THIS^.testValueIsNaN(THIS^.NAN);
THIS^.testValueIsNaN(THIS^.INF);
THIS^.testValueIsNaN(THIS^.MINUS_INF);
THIS^.testValueIsNaN(THIS^.MAX_NON_SPECIAL);
THIS^.testValueIsNaN(THIS^.MIN_NON_SPECIAL);
THIS^.testValueIsNaN(THIS^.ZERO);
THIS^.testValueIsNaN(THIS^.MINUS_ZERO);
THIS^.testValueIsNaN(THIS^.MAX_SUBNORMAL);
THIS^.testValueIsNaN(THIS^.MIN_SUBNORMAL);
THIS^.testValueIsNaN(THIS^.SMALLEST_NEGATIVE_SUBNORMAL);
THIS^.testValueIsNaN(THIS^.SMALLEST_POSITIVE_SUBNORMAL);
THIS^.testValueIsNaN(THIS^.ONE_PERCENT);
THIS^.testValueIsNaN(THIS^.ONE_PERMILLE);
THIS^.testValueIsNaN(THIS^.MINUS_ONE_PERCENT);
THIS^.testValueIsNaN(THIS^.MINUS_ONE_PERMILLE);

TcUnit.TEST_FINISHED();
END_METHOD

(*

short summary
==================
This test method tests ``assert.float.double.valueIsNegativeInfinite``
method of CNM_AssertionInterfaces library with various inputs

.. <legal notes>

legal notes
=================
| SPDX-FileCopyrightText: © 2022 ekvip automation GmbH <info@ekvip.de>
| SPDX-License-Identifier: Apache-2.0
| For details check: Apache-2.0_

.. _Apache-2.0: https://www.apache.org/licenses/LICENSE-2.0

.. </legal notes>

*)

METHOD runValueIsNegativeInfiniteTests
RETURN (NOT TcUnit.TEST_ORDERED(THIS^.getTestNameFor('valueIsNegativeInfinite')));

THIS^.testValueIsNegativeInfinite(THIS^.NAN);
THIS^.testValueIsNegativeInfinite(THIS^.INF);
THIS^.testValueIsNegativeInfinite(THIS^.MINUS_INF);
THIS^.testValueIsNegativeInfinite(THIS^.MAX_NON_SPECIAL);
THIS^.testValueIsNegativeInfinite(THIS^.MIN_NON_SPECIAL);
THIS^.testValueIsNegativeInfinite(THIS^.ZERO);
THIS^.testValueIsNegativeInfinite(THIS^.MINUS_ZERO);
THIS^.testValueIsNegativeInfinite(THIS^.MAX_SUBNORMAL);
THIS^.testValueIsNegativeInfinite(THIS^.MIN_SUBNORMAL);
THIS^.testValueIsNegativeInfinite(THIS^.SMALLEST_NEGATIVE_SUBNORMAL);
THIS^.testValueIsNegativeInfinite(THIS^.SMALLEST_POSITIVE_SUBNORMAL);
THIS^.testValueIsNegativeInfinite(THIS^.ONE_PERCENT);
THIS^.testValueIsNegativeInfinite(THIS^.ONE_PERMILLE);
THIS^.testValueIsNegativeInfinite(THIS^.MINUS_ONE_PERCENT);
THIS^.testValueIsNegativeInfinite(THIS^.MINUS_ONE_PERMILLE);

TcUnit.TEST_FINISHED();
END_METHOD

(*

short summary
==================
This test method tests ``assert.float.double.valueIsNegative``
method of CNM_AssertionInterfaces library with various inputs

.. <legal notes>

legal notes
=================
| SPDX-FileCopyrightText: © 2022 ekvip automation GmbH <info@ekvip.de>
| SPDX-License-Identifier: Apache-2.0
| For details check: Apache-2.0_

.. _Apache-2.0: https://www.apache.org/licenses/LICENSE-2.0

.. </legal notes>

*)

METHOD runValueIsNegativeTests
RETURN (NOT TcUnit.TEST_ORDERED(THIS^.getTestNameFor('valueIsNegative')));

THIS^.testValueIsNegative(THIS^.NAN);
THIS^.testValueIsNegative(THIS^.INF);
THIS^.testValueIsNegative(THIS^.MINUS_INF);
THIS^.testValueIsNegative(THIS^.MAX_NON_SPECIAL);
THIS^.testValueIsNegative(THIS^.MIN_NON_SPECIAL);
THIS^.testValueIsNegative(THIS^.ZERO);
THIS^.testValueIsNegative(THIS^.MINUS_ZERO);
THIS^.testValueIsNegative(THIS^.MAX_SUBNORMAL);
THIS^.testValueIsNegative(THIS^.MIN_SUBNORMAL);
THIS^.testValueIsNegative(THIS^.SMALLEST_NEGATIVE_SUBNORMAL);
THIS^.testValueIsNegative(THIS^.SMALLEST_POSITIVE_SUBNORMAL);
THIS^.testValueIsNegative(THIS^.ONE_PERCENT);
THIS^.testValueIsNegative(THIS^.ONE_PERMILLE);
THIS^.testValueIsNegative(THIS^.MINUS_ONE_PERCENT);
THIS^.testValueIsNegative(THIS^.MINUS_ONE_PERMILLE);

TcUnit.TEST_FINISHED();
END_METHOD

(*

short summary
==================
This test method tests ``assert.float.double.valueIsNegativeZero``
method of CNM_AssertionInterfaces library with various inputs

.. <legal notes>

legal notes
=================
| SPDX-FileCopyrightText: © 2022 ekvip automation GmbH <info@ekvip.de>
| SPDX-License-Identifier: Apache-2.0
| For details check: Apache-2.0_

.. _Apache-2.0: https://www.apache.org/licenses/LICENSE-2.0

.. </legal notes>

*)

METHOD runValueIsNegativeZeroTests
RETURN (NOT TcUnit.TEST_ORDERED(THIS^.getTestNameFor('valueIsNegativeZero')));

THIS^.testValueIsNegativeZero(THIS^.NAN);
THIS^.testValueIsNegativeZero(THIS^.INF);
THIS^.testValueIsNegativeZero(THIS^.MINUS_INF);
THIS^.testValueIsNegativeZero(THIS^.MAX_NON_SPECIAL);
THIS^.testValueIsNegativeZero(THIS^.MIN_NON_SPECIAL);
THIS^.testValueIsNegativeZero(THIS^.ZERO);
THIS^.testValueIsNegativeZero(THIS^.MINUS_ZERO);
THIS^.testValueIsNegativeZero(THIS^.MAX_SUBNORMAL);
THIS^.testValueIsNegativeZero(THIS^.MIN_SUBNORMAL);
THIS^.testValueIsNegativeZero(THIS^.SMALLEST_NEGATIVE_SUBNORMAL);
THIS^.testValueIsNegativeZero(THIS^.SMALLEST_POSITIVE_SUBNORMAL);
THIS^.testValueIsNegativeZero(THIS^.ONE_PERCENT);
THIS^.testValueIsNegativeZero(THIS^.ONE_PERMILLE);
THIS^.testValueIsNegativeZero(THIS^.MINUS_ONE_PERCENT);
THIS^.testValueIsNegativeZero(THIS^.MINUS_ONE_PERMILLE);

TcUnit.TEST_FINISHED();
END_METHOD

(*

short summary
==================
This test method tests ``assert.float.double.valueIsNormal``
method of CNM_AssertionInterfaces library with various inputs

.. <legal notes>

legal notes
=================
| SPDX-FileCopyrightText: © 2022 ekvip automation GmbH <info@ekvip.de>
| SPDX-License-Identifier: Apache-2.0
| For details check: Apache-2.0_

.. _Apache-2.0: https://www.apache.org/licenses/LICENSE-2.0

.. </legal notes>

*)

METHOD runValueIsNormalTests
RETURN (NOT TcUnit.TEST_ORDERED(THIS^.getTestNameFor('valueIsNormal')));

THIS^.testValueIsNormal(THIS^.NAN);
THIS^.testValueIsNormal(THIS^.INF);
THIS^.testValueIsNormal(THIS^.MINUS_INF);
THIS^.testValueIsNormal(THIS^.MAX_NON_SPECIAL);
THIS^.testValueIsNormal(THIS^.MIN_NON_SPECIAL);
THIS^.testValueIsNormal(THIS^.ZERO);
THIS^.testValueIsNormal(THIS^.MINUS_ZERO);
THIS^.testValueIsNormal(THIS^.MAX_SUBNORMAL);
THIS^.testValueIsNormal(THIS^.MIN_SUBNORMAL);
THIS^.testValueIsNormal(THIS^.SMALLEST_NEGATIVE_SUBNORMAL);
THIS^.testValueIsNormal(THIS^.SMALLEST_POSITIVE_SUBNORMAL);
THIS^.testValueIsNormal(THIS^.ONE_PERCENT);
THIS^.testValueIsNormal(THIS^.ONE_PERMILLE);
THIS^.testValueIsNormal(THIS^.MINUS_ONE_PERCENT);
THIS^.testValueIsNormal(THIS^.MINUS_ONE_PERMILLE);

TcUnit.TEST_FINISHED();
END_METHOD

(*

short summary
==================
This test method tests ``assert.float.double.valueIsNotEqualTo``
method of CNM_AssertionInterfaces library with various inputs

.. <legal notes>

legal notes
=================
| SPDX-FileCopyrightText: © 2022 ekvip automation GmbH <info@ekvip.de>
| SPDX-License-Identifier: Apache-2.0
| For details check: Apache-2.0_

.. _Apache-2.0: https://www.apache.org/licenses/LICENSE-2.0

.. </legal notes>

*)

METHOD runValueIsNotEqualToTests
RETURN (NOT TcUnit.TEST_ORDERED(THIS^.getTestNameFor('valueIsNotEqualTo')));

THIS^.testValueIsNotEqualTo(
	valueToTest := THIS^.NAN,
	unexpectedValue := THIS^.ONE_PERCENT,
	tolerance := THIS^.ONE_PERMILLE
);

THIS^.testValueIsNotEqualTo(
	valueToTest := THIS^.ONE_PERCENT,
	unexpectedValue := THIS^.NAN,
	tolerance := THIS^.ONE_PERMILLE
);

THIS^.testValueIsNotEqualTo(
	valueToTest := THIS^.ONE_PERCENT,
	unexpectedValue := THIS^.ONE_PERCENT,
	tolerance := THIS^.NAN
);

THIS^.testValueIsNotEqualTo(
	valueToTest := THIS^.NAN,
	unexpectedValue := THIS^.NAN,
	tolerance := THIS^.ONE_PERCENT
);

THIS^.testValueIsNotEqualTo(
	valueToTest := THIS^.NAN,
	unexpectedValue := THIS^.NAN,
	tolerance := THIS^.NAN
);

THIS^.testValueIsNotEqualTo(
	valueToTest := THIS^.INF,
	unexpectedValue := THIS^.ONE_PERCENT,
	tolerance := THIS^.ONE_PERMILLE
);

THIS^.testValueIsNotEqualTo(
	valueToTest := THIS^.ONE_PERCENT,
	unexpectedValue := THIS^.INF,
	tolerance := THIS^.ONE_PERMILLE
);

THIS^.testValueIsNotEqualTo(
	valueToTest := THIS^.ONE_PERCENT,
	unexpectedValue := THIS^.ONE_PERCENT,
	tolerance := THIS^.INF
);

THIS^.testValueIsNotEqualTo(
	valueToTest := THIS^.INF,
	unexpectedValue := THIS^.INF,
	tolerance := THIS^.ONE_PERCENT
);

THIS^.testValueIsNotEqualTo(
	valueToTest := THIS^.INF,
	unexpectedValue := THIS^.INF,
	tolerance := THIS^.INF
);

THIS^.testValueIsNotEqualTo(
	valueToTest := THIS^.INF,
	unexpectedValue := THIS^.MINUS_INF,
	tolerance := THIS^.INF
);

THIS^.testValueIsNotEqualTo(
	valueToTest := THIS^.MINUS_INF,
	unexpectedValue := THIS^.ONE_PERCENT,
	tolerance := THIS^.ONE_PERMILLE
);

THIS^.testValueIsNotEqualTo(
	valueToTest := THIS^.ONE_PERCENT,
	unexpectedValue := THIS^.MINUS_INF,
	tolerance := THIS^.ONE_PERMILLE
);

THIS^.testValueIsNotEqualTo(
	valueToTest := THIS^.ONE_PERCENT,
	unexpectedValue := THIS^.ONE_PERCENT,
	tolerance := THIS^.MINUS_INF
);

THIS^.testValueIsNotEqualTo(
	valueToTest := THIS^.MINUS_INF,
	unexpectedValue := THIS^.MINUS_INF,
	tolerance := THIS^.ONE_PERCENT
);

THIS^.testValueIsNotEqualTo(
	valueToTest := THIS^.MINUS_INF,
	unexpectedValue := THIS^.MINUS_INF,
	tolerance := THIS^.MINUS_INF
);

THIS^.testValueIsNotEqualTo(
	valueToTest := THIS^.INF,
	unexpectedValue := THIS^.MINUS_INF,
	tolerance := THIS^.INF
);

THIS^.testValueIsNotEqualTo(
	valueToTest := THIS^.MINUS_ZERO,
	unexpectedValue := THIS^.SMALLEST_POSITIVE_SUBNORMAL,
	tolerance := THIS^.ONE_PERMILLE
);

THIS^.testValueIsNotEqualTo(
	valueToTest := THIS^.SMALLEST_POSITIVE_SUBNORMAL,
	unexpectedValue := THIS^.MINUS_ZERO,
	tolerance := THIS^.ONE_PERMILLE
);

THIS^.testValueIsNotEqualTo(
	valueToTest := THIS^.SMALLEST_POSITIVE_SUBNORMAL,
	unexpectedValue := THIS^.SMALLEST_POSITIVE_SUBNORMAL,
	tolerance := THIS^.MINUS_ZERO
);

THIS^.testValueIsNotEqualTo(
	valueToTest := THIS^.MINUS_ZERO,
	unexpectedValue := THIS^.MINUS_ZERO,
	tolerance := THIS^.SMALLEST_POSITIVE_SUBNORMAL
);

THIS^.testValueIsNotEqualTo(
	valueToTest := THIS^.MINUS_ZERO,
	unexpectedValue := THIS^.MINUS_ZERO,
	tolerance := THIS^.MINUS_ZERO
);

THIS^.testValueIsNotEqualTo(
	valueToTest := THIS^.MINUS_ZERO,
	unexpectedValue := THIS^.ZERO,
	tolerance := THIS^.MINUS_ZERO
);

THIS^.testValueIsNotEqualTo(
	valueToTest := THIS^.ZERO,
	unexpectedValue := THIS^.SMALLEST_POSITIVE_SUBNORMAL,
	tolerance := THIS^.ONE_PERMILLE
);

THIS^.testValueIsNotEqualTo(
	valueToTest := THIS^.SMALLEST_POSITIVE_SUBNORMAL,
	unexpectedValue := THIS^.ZERO,
	tolerance := THIS^.ONE_PERMILLE
);

THIS^.testValueIsNotEqualTo(
	valueToTest := THIS^.SMALLEST_POSITIVE_SUBNORMAL,
	unexpectedValue := THIS^.SMALLEST_POSITIVE_SUBNORMAL,
	tolerance := THIS^.ZERO
);

THIS^.testValueIsNotEqualTo(
	valueToTest := THIS^.ZERO,
	unexpectedValue := THIS^.ZERO,
	tolerance := THIS^.SMALLEST_POSITIVE_SUBNORMAL
);

THIS^.testValueIsNotEqualTo(
	valueToTest := THIS^.ZERO,
	unexpectedValue := THIS^.ZERO,
	tolerance := THIS^.ZERO
);

THIS^.testValueIsNotEqualTo(
	valueToTest := THIS^.ZERO,
	unexpectedValue := THIS^.MINUS_ZERO,
	tolerance := THIS^.ZERO
);

THIS^.testValueIsNotEqualTo(
	valueToTest := THIS^.SMALLEST_POSITIVE_SUBNORMAL,
	unexpectedValue := THIS^.ONE_PERCENT,
	tolerance := THIS^.ONE_PERMILLE
);

THIS^.testValueIsNotEqualTo(
	valueToTest := THIS^.ONE_PERCENT,
	unexpectedValue := THIS^.SMALLEST_POSITIVE_SUBNORMAL,
	tolerance := THIS^.ONE_PERMILLE
);

THIS^.testValueIsNotEqualTo(
	valueToTest := THIS^.ONE_PERCENT,
	unexpectedValue := THIS^.ONE_PERCENT,
	tolerance := THIS^.SMALLEST_POSITIVE_SUBNORMAL
);

THIS^.testValueIsNotEqualTo(
	valueToTest := THIS^.SMALLEST_POSITIVE_SUBNORMAL,
	unexpectedValue := THIS^.SMALLEST_POSITIVE_SUBNORMAL,
	tolerance := THIS^.ONE_PERCENT
);

THIS^.testValueIsNotEqualTo(
	valueToTest := THIS^.SMALLEST_POSITIVE_SUBNORMAL,
	unexpectedValue := THIS^.SMALLEST_POSITIVE_SUBNORMAL,
	tolerance := THIS^.SMALLEST_POSITIVE_SUBNORMAL
);

THIS^.testValueIsNotEqualTo(
	valueToTest := THIS^.SMALLEST_POSITIVE_SUBNORMAL,
	unexpectedValue := THIS^.SMALLEST_NEGATIVE_SUBNORMAL,
	tolerance := THIS^.SMALLEST_POSITIVE_SUBNORMAL
);

THIS^.testValueIsNotEqualTo(
	valueToTest := THIS^.SMALLEST_NEGATIVE_SUBNORMAL,
	unexpectedValue := THIS^.ONE_PERCENT,
	tolerance := THIS^.ONE_PERMILLE
);

THIS^.testValueIsNotEqualTo(
	valueToTest := THIS^.ONE_PERCENT,
	unexpectedValue := THIS^.SMALLEST_NEGATIVE_SUBNORMAL,
	tolerance := THIS^.ONE_PERMILLE
);

THIS^.testValueIsNotEqualTo(
	valueToTest := THIS^.ONE_PERCENT,
	unexpectedValue := THIS^.ONE_PERCENT,
	tolerance := THIS^.SMALLEST_NEGATIVE_SUBNORMAL
);

THIS^.testValueIsNotEqualTo(
	valueToTest := THIS^.SMALLEST_NEGATIVE_SUBNORMAL,
	unexpectedValue := THIS^.SMALLEST_NEGATIVE_SUBNORMAL,
	tolerance := THIS^.ONE_PERCENT
);

THIS^.testValueIsNotEqualTo(
	valueToTest := THIS^.SMALLEST_NEGATIVE_SUBNORMAL,
	unexpectedValue := THIS^.SMALLEST_NEGATIVE_SUBNORMAL,
	tolerance := THIS^.SMALLEST_NEGATIVE_SUBNORMAL
);

THIS^.testValueIsNotEqualTo(
	valueToTest := THIS^.SMALLEST_NEGATIVE_SUBNORMAL,
	unexpectedValue := THIS^.SMALLEST_POSITIVE_SUBNORMAL,
	tolerance := THIS^.SMALLEST_NEGATIVE_SUBNORMAL
);

THIS^.testValueIsNotEqualTo(
	valueToTest := THIS^.MAX_SUBNORMAL,
	unexpectedValue := THIS^.SMALLEST_POSITIVE_SUBNORMAL,
	tolerance := THIS^.SMALLEST_NEGATIVE_SUBNORMAL
);

THIS^.testValueIsNotEqualTo(
	valueToTest := THIS^.SMALLEST_POSITIVE_SUBNORMAL,
	unexpectedValue := THIS^.MAX_SUBNORMAL,
	tolerance := THIS^.SMALLEST_NEGATIVE_SUBNORMAL
);

THIS^.testValueIsNotEqualTo(
	valueToTest := THIS^.SMALLEST_POSITIVE_SUBNORMAL,
	unexpectedValue := THIS^.SMALLEST_POSITIVE_SUBNORMAL,
	tolerance := THIS^.MAX_SUBNORMAL
);

THIS^.testValueIsNotEqualTo(
	valueToTest := THIS^.MAX_SUBNORMAL,
	unexpectedValue := THIS^.MAX_SUBNORMAL,
	tolerance := THIS^.SMALLEST_POSITIVE_SUBNORMAL
);

THIS^.testValueIsNotEqualTo(
	valueToTest := THIS^.MAX_SUBNORMAL,
	unexpectedValue := THIS^.MAX_SUBNORMAL,
	tolerance := THIS^.MAX_SUBNORMAL
);

THIS^.testValueIsNotEqualTo(
	valueToTest := THIS^.MAX_SUBNORMAL,
	unexpectedValue := THIS^.MIN_SUBNORMAL,
	tolerance := THIS^.MAX_SUBNORMAL
);
//
THIS^.testValueIsNotEqualTo(
	valueToTest := THIS^.MIN_SUBNORMAL,
	unexpectedValue := THIS^.SMALLEST_POSITIVE_SUBNORMAL,
	tolerance := THIS^.SMALLEST_NEGATIVE_SUBNORMAL
);

THIS^.testValueIsNotEqualTo(
	valueToTest := THIS^.SMALLEST_POSITIVE_SUBNORMAL,
	unexpectedValue := THIS^.MIN_SUBNORMAL,
	tolerance := THIS^.SMALLEST_NEGATIVE_SUBNORMAL
);

THIS^.testValueIsNotEqualTo(
	valueToTest := THIS^.SMALLEST_POSITIVE_SUBNORMAL,
	unexpectedValue := THIS^.SMALLEST_POSITIVE_SUBNORMAL,
	tolerance := THIS^.MIN_SUBNORMAL
);

THIS^.testValueIsNotEqualTo(
	valueToTest := THIS^.MIN_SUBNORMAL,
	unexpectedValue := THIS^.MIN_SUBNORMAL,
	tolerance := THIS^.SMALLEST_POSITIVE_SUBNORMAL
);

THIS^.testValueIsNotEqualTo(
	valueToTest := THIS^.MIN_SUBNORMAL,
	unexpectedValue := THIS^.MIN_SUBNORMAL,
	tolerance := THIS^.MIN_SUBNORMAL
);

THIS^.testValueIsNotEqualTo(
	valueToTest := THIS^.MIN_SUBNORMAL,
	unexpectedValue := THIS^.MAX_SUBNORMAL,
	tolerance := THIS^.MIN_SUBNORMAL
);

THIS^.testValueIsNotEqualTo(
	valueToTest := THIS^.MAX_NON_SPECIAL,
	unexpectedValue := THIS^.SMALLEST_POSITIVE_SUBNORMAL,
	tolerance := THIS^.SMALLEST_NEGATIVE_SUBNORMAL
);

THIS^.testValueIsNotEqualTo(
	valueToTest := THIS^.SMALLEST_POSITIVE_SUBNORMAL,
	unexpectedValue := THIS^.MAX_NON_SPECIAL,
	tolerance := THIS^.SMALLEST_NEGATIVE_SUBNORMAL
);

THIS^.testValueIsNotEqualTo(
	valueToTest := THIS^.SMALLEST_POSITIVE_SUBNORMAL,
	unexpectedValue := THIS^.SMALLEST_POSITIVE_SUBNORMAL,
	tolerance := THIS^.MAX_NON_SPECIAL
);

THIS^.testValueIsNotEqualTo(
	valueToTest := THIS^.MAX_NON_SPECIAL,
	unexpectedValue := THIS^.MAX_NON_SPECIAL,
	tolerance := THIS^.SMALLEST_POSITIVE_SUBNORMAL
);

THIS^.testValueIsNotEqualTo(
	valueToTest := THIS^.MAX_NON_SPECIAL,
	unexpectedValue := THIS^.MAX_NON_SPECIAL,
	tolerance := THIS^.MAX_NON_SPECIAL
);

THIS^.testValueIsNotEqualTo(
	valueToTest := THIS^.MAX_NON_SPECIAL,
	unexpectedValue := THIS^.MIN_NON_SPECIAL,
	tolerance := THIS^.MAX_NON_SPECIAL
);

THIS^.testValueIsNotEqualTo(
	valueToTest := THIS^.MIN_NON_SPECIAL,
	unexpectedValue := THIS^.SMALLEST_POSITIVE_SUBNORMAL,
	tolerance := THIS^.SMALLEST_NEGATIVE_SUBNORMAL
);

THIS^.testValueIsNotEqualTo(
	valueToTest := THIS^.SMALLEST_POSITIVE_SUBNORMAL,
	unexpectedValue := THIS^.MIN_NON_SPECIAL,
	tolerance := THIS^.SMALLEST_NEGATIVE_SUBNORMAL
);

THIS^.testValueIsNotEqualTo(
	valueToTest := THIS^.SMALLEST_POSITIVE_SUBNORMAL,
	unexpectedValue := THIS^.SMALLEST_POSITIVE_SUBNORMAL,
	tolerance := THIS^.MIN_NON_SPECIAL
);

THIS^.testValueIsNotEqualTo(
	valueToTest := THIS^.MIN_NON_SPECIAL,
	unexpectedValue := THIS^.MIN_NON_SPECIAL,
	tolerance := THIS^.SMALLEST_POSITIVE_SUBNORMAL
);

THIS^.testValueIsNotEqualTo(
	valueToTest := THIS^.MIN_NON_SPECIAL,
	unexpectedValue := THIS^.MIN_NON_SPECIAL,
	tolerance := THIS^.MIN_NON_SPECIAL
);

THIS^.testValueIsNotEqualTo(
	valueToTest := THIS^.MAX_NON_SPECIAL,
	unexpectedValue := THIS^.MIN_NON_SPECIAL,
	tolerance := THIS^.MAX_NON_SPECIAL
);

TcUnit.TEST_FINISHED();
END_METHOD

(*

short summary
==================
This test method tests ``assert.float.double.valueIsNotNegativeInfinite``
method of CNM_AssertionInterfaces library with various inputs

.. <legal notes>

legal notes
=================
| SPDX-FileCopyrightText: © 2022 ekvip automation GmbH <info@ekvip.de>
| SPDX-License-Identifier: Apache-2.0
| For details check: Apache-2.0_

.. _Apache-2.0: https://www.apache.org/licenses/LICENSE-2.0

.. </legal notes>

*)

METHOD runValueIsNotNegativeInfiniteTests
RETURN (NOT TcUnit.TEST_ORDERED(THIS^.getTestNameFor('valueIsNotNegativeInfinite')));

THIS^.testValueIsNotNegativeInfinite(THIS^.NAN);
THIS^.testValueIsNotNegativeInfinite(THIS^.INF);
THIS^.testValueIsNotNegativeInfinite(THIS^.MINUS_INF);
THIS^.testValueIsNotNegativeInfinite(THIS^.MAX_NON_SPECIAL);
THIS^.testValueIsNotNegativeInfinite(THIS^.MIN_NON_SPECIAL);
THIS^.testValueIsNotNegativeInfinite(THIS^.ZERO);
THIS^.testValueIsNotNegativeInfinite(THIS^.MINUS_ZERO);
THIS^.testValueIsNotNegativeInfinite(THIS^.MAX_SUBNORMAL);
THIS^.testValueIsNotNegativeInfinite(THIS^.MIN_SUBNORMAL);
THIS^.testValueIsNotNegativeInfinite(THIS^.SMALLEST_NEGATIVE_SUBNORMAL);
THIS^.testValueIsNotNegativeInfinite(THIS^.SMALLEST_POSITIVE_SUBNORMAL);
THIS^.testValueIsNotNegativeInfinite(THIS^.ONE_PERCENT);
THIS^.testValueIsNotNegativeInfinite(THIS^.ONE_PERMILLE);
THIS^.testValueIsNotNegativeInfinite(THIS^.MINUS_ONE_PERCENT);
THIS^.testValueIsNotNegativeInfinite(THIS^.MINUS_ONE_PERMILLE);

TcUnit.TEST_FINISHED();
END_METHOD

(*

short summary
==================
This test method tests ``assert.float.double.valueIsNotPositiveInfinite``
method of CNM_AssertionInterfaces library with various inputs

.. <legal notes>

legal notes
=================
| SPDX-FileCopyrightText: © 2022 ekvip automation GmbH <info@ekvip.de>
| SPDX-License-Identifier: Apache-2.0
| For details check: Apache-2.0_

.. _Apache-2.0: https://www.apache.org/licenses/LICENSE-2.0

.. </legal notes>

*)

METHOD runValueIsNotPositiveInfiniteTests
RETURN (NOT TcUnit.TEST_ORDERED(THIS^.getTestNameFor('valueIsNotPositiveInfinite')));

THIS^.testValueIsNotPositiveInfinite(THIS^.NAN);
THIS^.testValueIsNotPositiveInfinite(THIS^.INF);
THIS^.testValueIsNotPositiveInfinite(THIS^.MINUS_INF);
THIS^.testValueIsNotPositiveInfinite(THIS^.MAX_NON_SPECIAL);
THIS^.testValueIsNotPositiveInfinite(THIS^.MIN_NON_SPECIAL);
THIS^.testValueIsNotPositiveInfinite(THIS^.ZERO);
THIS^.testValueIsNotPositiveInfinite(THIS^.MINUS_ZERO);
THIS^.testValueIsNotPositiveInfinite(THIS^.MAX_SUBNORMAL);
THIS^.testValueIsNotPositiveInfinite(THIS^.MIN_SUBNORMAL);
THIS^.testValueIsNotPositiveInfinite(THIS^.SMALLEST_NEGATIVE_SUBNORMAL);
THIS^.testValueIsNotPositiveInfinite(THIS^.SMALLEST_POSITIVE_SUBNORMAL);
THIS^.testValueIsNotPositiveInfinite(THIS^.ONE_PERCENT);
THIS^.testValueIsNotPositiveInfinite(THIS^.ONE_PERMILLE);
THIS^.testValueIsNotPositiveInfinite(THIS^.MINUS_ONE_PERCENT);
THIS^.testValueIsNotPositiveInfinite(THIS^.MINUS_ONE_PERMILLE);

TcUnit.TEST_FINISHED();
END_METHOD

(*

short summary
==================
This test method tests ``assert.float.double.valueIsNotSpecial``
method of CNM_AssertionInterfaces library with various inputs

.. <legal notes>

legal notes
=================
| SPDX-FileCopyrightText: © 2022 ekvip automation GmbH <info@ekvip.de>
| SPDX-License-Identifier: Apache-2.0
| For details check: Apache-2.0_

.. _Apache-2.0: https://www.apache.org/licenses/LICENSE-2.0

.. </legal notes>

*)

METHOD runValueIsNotSpecialTests
RETURN (NOT TcUnit.TEST_ORDERED(THIS^.getTestNameFor('valueIsNotSpecial')));

THIS^.testValueIsNotSpecial(THIS^.NAN);
THIS^.testValueIsNotSpecial(THIS^.INF);
THIS^.testValueIsNotSpecial(THIS^.MINUS_INF);
THIS^.testValueIsNotSpecial(THIS^.MAX_NON_SPECIAL);
THIS^.testValueIsNotSpecial(THIS^.MIN_NON_SPECIAL);
THIS^.testValueIsNotSpecial(THIS^.ZERO);
THIS^.testValueIsNotSpecial(THIS^.MINUS_ZERO);
THIS^.testValueIsNotSpecial(THIS^.MAX_SUBNORMAL);
THIS^.testValueIsNotSpecial(THIS^.MIN_SUBNORMAL);
THIS^.testValueIsNotSpecial(THIS^.SMALLEST_NEGATIVE_SUBNORMAL);
THIS^.testValueIsNotSpecial(THIS^.SMALLEST_POSITIVE_SUBNORMAL);
THIS^.testValueIsNotSpecial(THIS^.ONE_PERCENT);
THIS^.testValueIsNotSpecial(THIS^.ONE_PERMILLE);
THIS^.testValueIsNotSpecial(THIS^.MINUS_ONE_PERCENT);
THIS^.testValueIsNotSpecial(THIS^.MINUS_ONE_PERMILLE);

TcUnit.TEST_FINISHED();
END_METHOD

(*

short summary
==================
This test method tests ``assert.float.double.valueIsPositiveInfinite``
method of CNM_AssertionInterfaces library with various inputs

.. <legal notes>

legal notes
=================
| SPDX-FileCopyrightText: © 2022 ekvip automation GmbH <info@ekvip.de>
| SPDX-License-Identifier: Apache-2.0
| For details check: Apache-2.0_

.. _Apache-2.0: https://www.apache.org/licenses/LICENSE-2.0

.. </legal notes>

*)

METHOD runValueIsPositiveInfiniteTests
RETURN (NOT TcUnit.TEST_ORDERED(THIS^.getTestNameFor('valueIsPositiveInfinite')));

THIS^.testValueIsPositiveInfinite(THIS^.NAN);
THIS^.testValueIsPositiveInfinite(THIS^.INF);
THIS^.testValueIsPositiveInfinite(THIS^.MINUS_INF);
THIS^.testValueIsPositiveInfinite(THIS^.MAX_NON_SPECIAL);
THIS^.testValueIsPositiveInfinite(THIS^.MIN_NON_SPECIAL);
THIS^.testValueIsPositiveInfinite(THIS^.ZERO);
THIS^.testValueIsPositiveInfinite(THIS^.MINUS_ZERO);
THIS^.testValueIsPositiveInfinite(THIS^.MAX_SUBNORMAL);
THIS^.testValueIsPositiveInfinite(THIS^.MIN_SUBNORMAL);
THIS^.testValueIsPositiveInfinite(THIS^.SMALLEST_NEGATIVE_SUBNORMAL);
THIS^.testValueIsPositiveInfinite(THIS^.SMALLEST_POSITIVE_SUBNORMAL);
THIS^.testValueIsPositiveInfinite(THIS^.ONE_PERCENT);
THIS^.testValueIsPositiveInfinite(THIS^.ONE_PERMILLE);
THIS^.testValueIsPositiveInfinite(THIS^.MINUS_ONE_PERCENT);
THIS^.testValueIsPositiveInfinite(THIS^.MINUS_ONE_PERMILLE);

TcUnit.TEST_FINISHED();
END_METHOD

(*

short summary
==================
This test method tests ``assert.float.double.valueIsPositive``
method of CNM_AssertionInterfaces library with various inputs

.. <legal notes>

legal notes
=================
| SPDX-FileCopyrightText: © 2022 ekvip automation GmbH <info@ekvip.de>
| SPDX-License-Identifier: Apache-2.0
| For details check: Apache-2.0_

.. _Apache-2.0: https://www.apache.org/licenses/LICENSE-2.0

.. </legal notes>

*)

METHOD runValueIsPositiveTests
RETURN (NOT TcUnit.TEST_ORDERED(THIS^.getTestNameFor('valueIsPositive')));

THIS^.testValueIsPositive(THIS^.NAN);
THIS^.testValueIsPositive(THIS^.INF);
THIS^.testValueIsPositive(THIS^.MINUS_INF);
THIS^.testValueIsPositive(THIS^.MAX_NON_SPECIAL);
THIS^.testValueIsPositive(THIS^.MIN_NON_SPECIAL);
THIS^.testValueIsPositive(THIS^.ZERO);
THIS^.testValueIsPositive(THIS^.MINUS_ZERO);
THIS^.testValueIsPositive(THIS^.MAX_SUBNORMAL);
THIS^.testValueIsPositive(THIS^.MIN_SUBNORMAL);
THIS^.testValueIsPositive(THIS^.SMALLEST_NEGATIVE_SUBNORMAL);
THIS^.testValueIsPositive(THIS^.SMALLEST_POSITIVE_SUBNORMAL);
THIS^.testValueIsPositive(THIS^.ONE_PERCENT);
THIS^.testValueIsPositive(THIS^.ONE_PERMILLE);
THIS^.testValueIsPositive(THIS^.MINUS_ONE_PERCENT);
THIS^.testValueIsPositive(THIS^.MINUS_ONE_PERMILLE);

TcUnit.TEST_FINISHED();
END_METHOD

(*

short summary
==================
This test method tests ``assert.float.double.valueIsPositiveZero``
method of CNM_AssertionInterfaces library with various inputs

.. <legal notes>

legal notes
=================
| SPDX-FileCopyrightText: © 2022 ekvip automation GmbH <info@ekvip.de>
| SPDX-License-Identifier: Apache-2.0
| For details check: Apache-2.0_

.. _Apache-2.0: https://www.apache.org/licenses/LICENSE-2.0

.. </legal notes>

*)

METHOD runValueIsPositiveZeroTests
RETURN (NOT TcUnit.TEST_ORDERED(THIS^.getTestNameFor('valueIsPositiveZero')));

THIS^.testValueIsPositiveZero(THIS^.NAN);
THIS^.testValueIsPositiveZero(THIS^.INF);
THIS^.testValueIsPositiveZero(THIS^.MINUS_INF);
THIS^.testValueIsPositiveZero(THIS^.MAX_NON_SPECIAL);
THIS^.testValueIsPositiveZero(THIS^.MIN_NON_SPECIAL);
THIS^.testValueIsPositiveZero(THIS^.ZERO);
THIS^.testValueIsPositiveZero(THIS^.MINUS_ZERO);
THIS^.testValueIsPositiveZero(THIS^.MAX_SUBNORMAL);
THIS^.testValueIsPositiveZero(THIS^.MIN_SUBNORMAL);
THIS^.testValueIsPositiveZero(THIS^.SMALLEST_NEGATIVE_SUBNORMAL);
THIS^.testValueIsPositiveZero(THIS^.SMALLEST_POSITIVE_SUBNORMAL);
THIS^.testValueIsPositiveZero(THIS^.ONE_PERCENT);
THIS^.testValueIsPositiveZero(THIS^.ONE_PERMILLE);
THIS^.testValueIsPositiveZero(THIS^.MINUS_ONE_PERCENT);
THIS^.testValueIsPositiveZero(THIS^.MINUS_ONE_PERMILLE);

TcUnit.TEST_FINISHED();
END_METHOD

(*

short summary
==================
This test method tests ``assert.float.double.valueIsSpecial``
method of CNM_AssertionInterfaces library with various inputs

.. <legal notes>

legal notes
=================
| SPDX-FileCopyrightText: © 2022 ekvip automation GmbH <info@ekvip.de>
| SPDX-License-Identifier: Apache-2.0
| For details check: Apache-2.0_

.. _Apache-2.0: https://www.apache.org/licenses/LICENSE-2.0

.. </legal notes>

*)

METHOD runValueIsSpecialTests
RETURN (NOT TcUnit.TEST_ORDERED(THIS^.getTestNameFor('valueIsSpecial')));

THIS^.testValueIsSpecial(THIS^.NAN);
THIS^.testValueIsSpecial(THIS^.INF);
THIS^.testValueIsSpecial(THIS^.MINUS_INF);
THIS^.testValueIsSpecial(THIS^.MAX_NON_SPECIAL);
THIS^.testValueIsSpecial(THIS^.MIN_NON_SPECIAL);
THIS^.testValueIsSpecial(THIS^.ZERO);
THIS^.testValueIsSpecial(THIS^.MINUS_ZERO);
THIS^.testValueIsSpecial(THIS^.MAX_SUBNORMAL);
THIS^.testValueIsSpecial(THIS^.MIN_SUBNORMAL);
THIS^.testValueIsSpecial(THIS^.SMALLEST_NEGATIVE_SUBNORMAL);
THIS^.testValueIsSpecial(THIS^.SMALLEST_POSITIVE_SUBNORMAL);
THIS^.testValueIsSpecial(THIS^.ONE_PERCENT);
THIS^.testValueIsSpecial(THIS^.ONE_PERMILLE);
THIS^.testValueIsSpecial(THIS^.MINUS_ONE_PERCENT);
THIS^.testValueIsSpecial(THIS^.MINUS_ONE_PERMILLE);

TcUnit.TEST_FINISHED();
END_METHOD

(*

short summary
==================
This test method tests ``assert.float.double.valueIsSubnormal``
method of CNM_AssertionInterfaces library with various inputs

.. <legal notes>

legal notes
=================
| SPDX-FileCopyrightText: © 2022 ekvip automation GmbH <info@ekvip.de>
| SPDX-License-Identifier: Apache-2.0
| For details check: Apache-2.0_

.. _Apache-2.0: https://www.apache.org/licenses/LICENSE-2.0

.. </legal notes>

*)

METHOD runValueIsSubnormalTests
RETURN (NOT TcUnit.TEST_ORDERED(THIS^.getTestNameFor('valueIsSubnormal')));

THIS^.testValueIsSubnormal(THIS^.NAN);
THIS^.testValueIsSubnormal(THIS^.INF);
THIS^.testValueIsSubnormal(THIS^.MINUS_INF);
THIS^.testValueIsSubnormal(THIS^.MAX_NON_SPECIAL);
THIS^.testValueIsSubnormal(THIS^.MIN_NON_SPECIAL);
THIS^.testValueIsSubnormal(THIS^.ZERO);
THIS^.testValueIsSubnormal(THIS^.MINUS_ZERO);
THIS^.testValueIsSubnormal(THIS^.MAX_SUBNORMAL);
THIS^.testValueIsSubnormal(THIS^.MIN_SUBNORMAL);
THIS^.testValueIsSubnormal(THIS^.SMALLEST_NEGATIVE_SUBNORMAL);
THIS^.testValueIsSubnormal(THIS^.SMALLEST_POSITIVE_SUBNORMAL);
THIS^.testValueIsSubnormal(THIS^.ONE_PERCENT);
THIS^.testValueIsSubnormal(THIS^.ONE_PERMILLE);
THIS^.testValueIsSubnormal(THIS^.MINUS_ONE_PERCENT);
THIS^.testValueIsSubnormal(THIS^.MINUS_ONE_PERMILLE);

TcUnit.TEST_FINISHED();
END_METHOD

(*

short summary
==================
This test method tests ``assert.float.double.valueIsANumber``
method of CNM_AssertionInterfaces library, 
it provides the possibility to handover test data via parameter 

.. <legal notes>

legal notes
=================
| SPDX-FileCopyrightText: © 2022 ekvip automation GmbH <info@ekvip.de>
| SPDX-License-Identifier: Apache-2.0
| For details check: Apache-2.0_

.. _Apache-2.0: https://www.apache.org/licenses/LICENSE-2.0

.. </legal notes>

parameters
==========

*)

METHOD testValueIsANumber
VAR_INPUT
	(* for the test it's the parameter ``currentValue`` *)
	valueToTest	:LRealTestParameter;	
END_VAR
VAR
	(* just the expectation if the assertion to test must be worng or true *)
	assertionIsWrong		:BOOL;
	(* contains the format string for the test message *)
	message					:Tc2_System.T_MaxString;
	(* TwinCAT printf with the test message *)
	messageStringBuilder	:Tc2_Utilities.FB_FormatString;
	(* value of the paramter ``valueToTest`` as string *)
	valueToTestAsString		:Tc2_System.T_MaxString;
END_VAR
THIS^.assertorContainer.resetAssertor();

assertionIsWrong := Tc2_Utilities.LrealIsNaN(valueToTest.value);

message := SEL(
	assertionIsWrong,
	'currentValue is %s assertion must be TRUE', 
	'currentValue is %s assertion must be FALSE'
);

valueToTestAsString := valueToTest.asString;

messageStringBuilder(
	sFormat := message,
	arg1 := THIS^.AnyToArg(valueToTestAsString)
);

THIS^.assertorContainer.assertor.assert.float.double.valueIsANumber(
	currentValue := valueToTest.value,
	message := ''
);

THIS^.AssertEquals_BOOL(
	Expected 	:= assertionIsWrong,
	Actual 		:= THIS^.assertorContainer.wasAssertionWrong,
	Message 	:= messageStringBuilder.sOut
);
END_METHOD

(*

short summary
==================
This test method tests ``assert.float.double.valueIsEqualTo``
method of CNM_AssertionInterfaces library, 
it provides the possibility to handover test data via parameter 


.. <legal notes>

legal notes
=================
| SPDX-FileCopyrightText: © 2022 ekvip automation GmbH <info@ekvip.de>
| SPDX-License-Identifier: Apache-2.0
| For details check: Apache-2.0_

.. _Apache-2.0: https://www.apache.org/licenses/LICENSE-2.0

.. </legal notes>

parameters
==========

*)

METHOD testValueIsEqualTo 
VAR_INPUT
	(* for the test it's the parameter ``currentValue`` *)
	valueToTest	:LRealTestParameter;
	(* for the test it's the parameter ``expectedValue`` *)
	expected	:LRealTestParameter;
	(* for the test it's the parameter ``tolerance`` *)
	tolerance	:LRealTestParameter;
END_VAR
VAR
	(* just the expectation if the assertion to test must be worng or true *)
	assertionIsWrong		:BOOL;
	(* contains the format string for the test message *)
	message					:Tc2_System.T_MaxString;
	(* TwinCAT printf with the test message *)
	messageStringBuilder	:Tc2_Utilities.FB_FormatString;
	(* just to cast *)
	binaryCurrentValue		:POINTER TO LWORD;
	(* just to cast *)
	binaryExpectedValue		:POINTER TO LWORD;
	(* value of the paramter ``valueToTest`` as string *)
	valueToTestAsString		:Tc2_System.T_MaxString;
	(* value of the paramter ``expected`` as string *)
	expectedAsString		:Tc2_System.T_MaxString;
	(* value of the paramter ``tolerance`` as string *)
	toleranceAsString		:Tc2_System.T_MaxString;	
END_VAR
THIS^.assertorContainer.resetAssertor();
IF (
	Tc2_Utilities.LrealIsNaN(valueToTest.value)
	OR Tc2_Utilities.LrealIsNaN(expected.value)
	OR Tc2_Utilities.LrealIsNaN(tolerance.value)
) THEN
	assertionIsWrong := TRUE;
ELSIF (NOT Tc2_Utilities.LrealIsFinite(tolerance.value)) THEN
	assertionIsWrong := FALSE;
ELSIF (Tc2_Utilities.LrealIsFinite(valueToTest.value) <> Tc2_Utilities.LrealIsFinite(expected.value)) THEN
	assertionIsWrong := TRUE; 
ELSIF (
	(NOT Tc2_Utilities.LrealIsFinite(valueToTest.value))
	OR (NOT Tc2_Utilities.LrealIsFinite(expected.value))
) THEN
	binaryCurrentValue := ADR(valueToTest.value);
	binaryExpectedValue := ADR(expected.value);
	assertionIsWrong := (binaryCurrentValue^.SIGN <> binaryExpectedValue^.SIGN);
ELSE
	assertionIsWrong := (
		((expected.value + ABS(tolerance.value)) < valueToTest.value)
		OR ((expected.value - ABS(tolerance.value)) > valueToTest.value)
	);
END_IF

message := SEL(
	assertionIsWrong,
	'currentValue is %s expectedValue is %s tolerance is %s assertion must be TRUE', 
	'currentValue is %s expectedValue is %s tolerance is %s assertion must be FALSE'
);

valueToTestAsString := valueToTest.asString;
expectedAsString := expected.asString;
toleranceAsString := tolerance.asString;

messageStringBuilder(
	sFormat := message,
	arg1 := THIS^.AnyToArg(valueToTestAsString),
	arg2 := THIS^.AnyToArg(expectedAsString),
	arg3 := THIS^.AnyToArg(toleranceAsString)
);

THIS^.assertorContainer.assertor.assert.float.double.valueIsEqualTo(
	currentValue	:= valueToTest.value,
	expectedValue	:= expected.value,
	tolerance       := tolerance.value,
	message			:= ''
);

THIS^.AssertEquals_BOOL(
	Expected 	:= assertionIsWrong,
	Actual 		:= THIS^.assertorContainer.wasAssertionWrong,
	Message 	:= messageStringBuilder.sOut
);
END_METHOD

(*

short summary
==================
This test method tests ``assert.float.double.valueIsFinite``
method of CNM_AssertionInterfaces library, 
it provides the possibility to handover test data via parameter 

.. <legal notes>

legal notes
=================
| SPDX-FileCopyrightText: © 2022 ekvip automation GmbH <info@ekvip.de>
| SPDX-License-Identifier: Apache-2.0
| For details check: Apache-2.0_

.. _Apache-2.0: https://www.apache.org/licenses/LICENSE-2.0

.. </legal notes>

parameters
==========

*)

METHOD testValueIsFinite
VAR_INPUT
	(* for the test it's the parameter ``currentValue`` *)
	valueToTest	:LRealTestParameter;	
END_VAR
VAR
	(* just the expectation if the assertion to test must be worng or true *)
	assertionIsWrong		:BOOL;
	(* contains the format string for the test message *)
	message					:Tc2_System.T_MaxString;
	(* TwinCAT printf with the test message *)
	messageStringBuilder	:Tc2_Utilities.FB_FormatString;
	(* value of the paramter ``valueToTest`` as string *)
	valueToTestAsString		:Tc2_System.T_MaxString;
	(* binary value of the parameter ``valueToTest`` *)
	binaryValueToTest		:POINTER TO LWORD;
END_VAR
THIS^.assertorContainer.resetAssertor();

binaryValueToTest := ADR(valueToTest.value);
assertionIsWrong := (
	(binaryValueToTest^ = THIS^.BINARY_INFINITY)
	OR_ELSE (binaryValueToTest^ = THIS^.BINARY_NEGATIVE_INFINITY)
);

message := SEL(
	assertionIsWrong,
	'currentValue is %s assertion must be TRUE', 
	'currentValue is %s assertion must be FALSE'
);

valueToTestAsString := valueToTest.asString;

messageStringBuilder(
	sFormat := message,
	arg1 := THIS^.AnyToArg(valueToTestAsString)
);

THIS^.assertorContainer.assertor.assert.float.double.valueIsFinite(
	currentValue := valueToTest.value,
	message := ''
);

THIS^.AssertEquals_BOOL(
	Expected 	:= assertionIsWrong,
	Actual 		:= THIS^.assertorContainer.wasAssertionWrong,
	Message 	:= messageStringBuilder.sOut
);
END_METHOD

(*

short summary
==================
This test method tests ``assert.float.double.valueIsGreaterThan``
method of CNM_AssertionInterfaces library, 
it provides the possibility to handover test data via parameter 


.. <legal notes>

legal notes
=================
| SPDX-FileCopyrightText: © 2022 ekvip automation GmbH <info@ekvip.de>
| SPDX-License-Identifier: Apache-2.0
| For details check: Apache-2.0_

.. _Apache-2.0: https://www.apache.org/licenses/LICENSE-2.0

.. </legal notes>

parameters
==========

*)

METHOD testValueIsGreaterThan 
VAR_INPUT
	(* for the test it's the parameter ``currentValue`` *)
	valueToTest	:LRealTestParameter;
	(* for the test it's the parameter ``lessValue`` *)
	lessValue	:LRealTestParameter;
END_VAR
VAR
	(* just the expectation if the assertion to test must be worng or true *)
	assertionIsWrong		:BOOL;
	(* contains the format string for the test message *)
	message					:Tc2_System.T_MaxString;
	(* TwinCAT printf with the test message *)
	messageStringBuilder	:Tc2_Utilities.FB_FormatString;
	(* just to cast *)
	binaryCurrentValue		:POINTER TO LWORD;
	(* just to cast *)
	binaryLessValue			:POINTER TO LWORD;
	(* value of the paramter ``valueToTest`` as string *)
	valueToTestAsString		:Tc2_System.T_MaxString;
	(* value of the paramter ``lessValue`` as string *)
	lessValueAsString		:Tc2_System.T_MaxString;	
END_VAR
THIS^.assertorContainer.resetAssertor();

IF (Tc2_Utilities.LrealIsNaN(valueToTest.value) OR Tc2_Utilities.LrealIsNaN(lessValue.value)) THEN
	assertionIsWrong := TRUE;
ELSIF ((NOT Tc2_Utilities.LrealIsFinite(valueToTest.value)) AND (NOT Tc2_Utilities.LrealIsFinite(lessValue.value))) THEN
	binaryCurrentValue := ADR(valueToTest.value);
	binaryLessValue := ADR(lessValue.value);
	assertionIsWrong := (
		(binaryCurrentValue^.SIGN) //-inf
		OR (NOT binaryLessValue^.SIGN) //inf
	);
ELSIF ((NOT Tc2_Utilities.LrealIsFinite(valueToTest.value)) AND (Tc2_Utilities.LrealIsFinite(lessValue.value))) THEN
	binaryCurrentValue := ADR(valueToTest.value);
	assertionIsWrong := (binaryCurrentValue^.SIGN);
ELSIF (
	(Tc2_Utilities.LrealIsFinite(valueToTest.value))
	AND (NOT Tc2_Utilities.LrealIsFinite(lessValue.value))
) THEN
	binaryLessValue := ADR(lessValue.value);
	assertionIsWrong := (NOT binaryLessValue^.SIGN);
ELSE
	assertionIsWrong := (valueToTest.value <= lessValue.value);
END_IF

message := SEL(
	assertionIsWrong,
	'currentValue is %s lessValue is %s assertion must be TRUE', 
	'currentValue is %s lessValue is %s assertion must be FALSE'
);

valueToTestAsString := valueToTest.asString;
lessValueAsString := lessValue.asString;

messageStringBuilder(
	sFormat := message,
	arg1 := THIS^.AnyToArg(valueToTestAsString),
	arg2 := THIS^.AnyToArg(lessValueAsString)
);

THIS^.assertorContainer.assertor.assert.float.double.valueIsGreaterThan(
	currentValue	:= valueToTest.value,
	lessValue		:= lessValue.value,
	message			:= ''
);

THIS^.AssertEquals_BOOL(
	Expected 	:= assertionIsWrong,
	Actual 		:= THIS^.assertorContainer.wasAssertionWrong,
	Message 	:= messageStringBuilder.sOut
);
END_METHOD

(*

short summary
==================
This test method tests ``assert.float.double.valueIsInfinite``
method of CNM_AssertionInterfaces library, 
it provides the possibility to handover test data via parameter 

.. <legal notes>

legal notes
=================
| SPDX-FileCopyrightText: © 2022 ekvip automation GmbH <info@ekvip.de>
| SPDX-License-Identifier: Apache-2.0
| For details check: Apache-2.0_

.. _Apache-2.0: https://www.apache.org/licenses/LICENSE-2.0

.. </legal notes>

parameters
==========

*)

METHOD testValueIsInfinite
VAR_INPUT
	(* for the test it's the parameter ``currentValue`` *)
	valueToTest	:LRealTestParameter;	
END_VAR
VAR
	(* just the expectation if the assertion to test must be worng or true *)
	assertionIsWrong		:BOOL;
	(* contains the format string for the test message *)
	message					:Tc2_System.T_MaxString;
	(* TwinCAT printf with the test message *)
	messageStringBuilder	:Tc2_Utilities.FB_FormatString;
	(* value of the paramter ``valueToTest`` as string *)
	valueToTestAsString		:Tc2_System.T_MaxString;
	(* binary value of the parameter ``valueToTest`` *)
	binaryValueToTest		:POINTER TO LWORD;
END_VAR
THIS^.assertorContainer.resetAssertor();

binaryValueToTest := ADR(valueToTest.value);
assertionIsWrong := (
	(binaryValueToTest^ <> THIS^.BINARY_INFINITY)
	AND_THEN (binaryValueToTest^ <> THIS^.BINARY_NEGATIVE_INFINITY)
);

message := SEL(
	assertionIsWrong,
	'currentValue is %s assertion must be TRUE', 
	'currentValue is %s assertion must be FALSE'
);

valueToTestAsString := valueToTest.asString;

messageStringBuilder(
	sFormat := message,
	arg1 := THIS^.AnyToArg(valueToTestAsString)
);

THIS^.assertorContainer.assertor.assert.float.double.valueIsInfinite(
	currentValue := valueToTest.value,
	message := ''
);

THIS^.AssertEquals_BOOL(
	Expected 	:= assertionIsWrong,
	Actual 		:= THIS^.assertorContainer.wasAssertionWrong,
	Message 	:= messageStringBuilder.sOut
);
END_METHOD

(*

short summary
==================
This test method tests ``assert.float.double.valueIsInRangeOf``
method of CNM_AssertionInterfaces library, 
it provides the possibility to handover test data via parameter 


.. <legal notes>

legal notes
=================
| SPDX-FileCopyrightText: © 2022 ekvip automation GmbH <info@ekvip.de>
| SPDX-License-Identifier: Apache-2.0
| For details check: Apache-2.0_

.. _Apache-2.0: https://www.apache.org/licenses/LICENSE-2.0

.. </legal notes>

parameters
==========

*)

METHOD testValueIsInRangeOf 
VAR_INPUT
	(* for the test it's the parameter ``lowerLimit`` *)
	lowerLimit	:LRealTestParameter;
	(* for the test it's the parameter ``currentValue`` *)
	valueToTest	:LRealTestParameter;
	(* for the test it's the parameter ``upperLimit`` *)
	upperLimit	:LRealTestParameter;
END_VAR
VAR
	(* just the expectation if the assertion to test must be worng or true *)
	assertionIsWrong		:BOOL;
	(* contains the format string for the test message *)
	message					:Tc2_System.T_MaxString;
	(* TwinCAT printf with the test message *)
	messageStringBuilder	:Tc2_Utilities.FB_FormatString;
	(* just to cast *)
	binaryLowerLimit		:POINTER TO LWORD;
	(* just to cast *)
	binaryCurrentValue		:POINTER TO LWORD;
	(* just to cast *)
	binaryUpperLimit		:POINTER TO LWORD;
	(* value of the paramter ``lowerLimit`` as string *)
	lowerLimitAsString		:Tc2_System.T_MaxString;
	(* value of the paramter ``valueToTest`` as string *)
	valueToTestAsString		:Tc2_System.T_MaxString;
	(* value of the paramter ``upperLimit`` as string *)
	upperLimitAsString		:Tc2_System.T_MaxString;	
END_VAR
THIS^.assertorContainer.resetAssertor();

IF (
	Tc2_Utilities.LrealIsNaN(lowerLimit.value)
	OR Tc2_Utilities.LrealIsNaN(valueToTest.value)
	OR  Tc2_Utilities.LrealIsNaN(upperLimit.value)
) THEN
	assertionIsWrong := TRUE;
ELSIF (
	(NOT Tc2_Utilities.LrealIsFinite(lowerLimit.value))
	AND (NOT Tc2_Utilities.LrealIsFinite(valueToTest.value))
	AND (NOT Tc2_Utilities.LrealIsFinite(upperLimit.value))
) THEN
	binaryLowerLimit	:= ADR(lowerLimit.value);
	binaryCurrentValue	:= ADR(valueToTest.value);
	binaryUpperLimit	:= ADR(upperLimit.value);
	assertionIsWrong := (
		((NOT binaryLowerLimit^.SIGN) AND binaryUpperLimit^.SIGN)
		OR (
			((NOT binaryLowerLimit^.SIGN) AND (NOT binaryUpperLimit^.SIGN) AND binaryCurrentValue^.SIGN)
		) OR (
			(binaryLowerLimit^.SIGN AND binaryUpperLimit^.SIGN AND (NOT binaryCurrentValue^.SIGN))
		)
	);
ELSIF (
	(Tc2_Utilities.LrealIsFinite(lowerLimit.value))
	AND (NOT Tc2_Utilities.LrealIsFinite(valueToTest.value))
	AND (Tc2_Utilities.LrealIsFinite(upperLimit.value))
) THEN
	assertionIsWrong := TRUE;
ELSIF (
	(NOT Tc2_Utilities.LrealIsFinite(lowerLimit.value))
	AND (Tc2_Utilities.LrealIsFinite(valueToTest.value))
	AND (Tc2_Utilities.LrealIsFinite(upperLimit.value))
) THEN
	binaryLowerLimit	:= ADR(lowerLimit.value);
	assertionIsWrong := (
		(NOT binaryLowerLimit^.SIGN)
		OR (valueToTest.value > upperLimit.value)
	);
ELSIF (
	(Tc2_Utilities.LrealIsFinite(lowerLimit.value))
	AND (Tc2_Utilities.LrealIsFinite(valueToTest.value))
	AND (NOT Tc2_Utilities.LrealIsFinite(upperLimit.value))
) THEN
	binaryUpperLimit	:= ADR(upperLimit.value);
	assertionIsWrong := (
		(binaryUpperLimit^.SIGN)
		OR (valueToTest.value < lowerLimit.value)
	);
ELSE
	assertionIsWrong := assertionIsWrong := (
		(valueToTest.value < lowerLimit.value)
		 OR (valueToTest.value > upperLimit.value)
	);
END_IF

message := SEL(
	assertionIsWrong,
	'lowerLimit is %s currentValue is %s upperLimit is %s assertion must be TRUE', 
	'lowerLimit is %s currentValue is %s upperLimit is %s assertion must be FALSE'
);

lowerLimitAsString	:= lowerLimit.asString;
valueToTestAsString := valueToTest.asString;
upperLimitAsString  := upperLimit.asString;

messageStringBuilder(
	sFormat := message,
	arg1 := THIS^.AnyToArg(lowerLimitAsString),
	arg2 := THIS^.AnyToArg(valueToTestAsString),
	arg3 := THIS^.AnyToArg(upperLimitAsString)
);

THIS^.assertorContainer.assertor.assert.float.double.valueIsInRangeOf(
	lowerLimit		:= lowerLimit.value,
	currentValue	:= valueToTest.value,
	upperLimit		:= upperLimit.value,
	message			:= ''
);

THIS^.AssertEquals_BOOL(
	Expected 	:= assertionIsWrong,
	Actual 		:= THIS^.assertorContainer.wasAssertionWrong,
	Message 	:= messageStringBuilder.sOut
);
END_METHOD

(*

short summary
==================
This test method tests ``assert.float.double.valueIsLessThan``
method of CNM_AssertionInterfaces library, 
it provides the possibility to handover test data via parameter 


.. <legal notes>

legal notes
=================
| SPDX-FileCopyrightText: © 2022 ekvip automation GmbH <info@ekvip.de>
| SPDX-License-Identifier: Apache-2.0
| For details check: Apache-2.0_

.. _Apache-2.0: https://www.apache.org/licenses/LICENSE-2.0

.. </legal notes>

parameters
==========

*)

METHOD testValueIsLessThan 
VAR_INPUT
	(* for the test it's the parameter ``currentValue`` *)
	valueToTest		:LRealTestParameter;
	(* for the test it's the parameter ``greaterValue`` *)
	greaterValue	:LRealTestParameter;
END_VAR
VAR
	(* just the expectation if the assertion to test must be worng or true *)
	assertionIsWrong		:BOOL;
	(* contains the format string for the test message *)
	message					:Tc2_System.T_MaxString;
	(* TwinCAT printf with the test message *)
	messageStringBuilder	:Tc2_Utilities.FB_FormatString;
	(* just to cast *)
	binaryCurrentValue		:POINTER TO LWORD;
	(* just to cast *)
	binaryGreaterValue		:POINTER TO LWORD;
	(* value of the paramter ``valueToTest`` as string *)
	valueToTestAsString		:Tc2_System.T_MaxString;
	(* value of the paramter ``greaterValue`` as string *)
	greaterValueAsString	:Tc2_System.T_MaxString;	
END_VAR
THIS^.assertorContainer.resetAssertor();

IF (
	Tc2_Utilities.LrealIsNaN(valueToTest.value) 
	OR Tc2_Utilities.LrealIsNaN(greaterValue.value)
) THEN
	assertionIsWrong := TRUE;
ELSIF (
	(NOT Tc2_Utilities.LrealIsFinite(valueToTest.value))
	AND (NOT Tc2_Utilities.LrealIsFinite(greaterValue.value))
) THEN
	binaryCurrentValue := ADR(valueToTest.value);
	binaryGreaterValue := ADR(greaterValue.value);
	assertionIsWrong := (
		(NOT binaryCurrentValue^.SIGN) //inf
		OR (binaryGreaterValue^.SIGN) //-inf
	);
ELSIF (
	(NOT Tc2_Utilities.LrealIsFinite(valueToTest.value))
	AND (Tc2_Utilities.LrealIsFinite(greaterValue.value))
) THEN
	binaryCurrentValue := ADR(valueToTest.value);
	assertionIsWrong := (NOT binaryCurrentValue^.SIGN); //inf
ELSIF (
	(Tc2_Utilities.LrealIsFinite(valueToTest.value))
	AND (NOT Tc2_Utilities.LrealIsFinite(greaterValue.value))
) THEN
	binaryGreaterValue := ADR(greaterValue.value);
	assertionIsWrong := (binaryGreaterValue^.SIGN); //-inf
ELSE
	assertionIsWrong := (valueToTest.value >= greaterValue.value);
END_IF

message := SEL(
	assertionIsWrong,
	'currentValue is %s greaterValue is %s assertion must be TRUE', 
	'currentValue is %s greaterValue is %s assertion must be FALSE'
);

valueToTestAsString := valueToTest.asString;
greaterValueAsString := greaterValue.asString;

messageStringBuilder(
	sFormat := message,
	arg1 := THIS^.AnyToArg(valueToTestAsString),
	arg2 := THIS^.AnyToArg(greaterValueAsString)
);

THIS^.assertorContainer.assertor.assert.float.double.valueIsLessThan(
	currentValue	:= valueToTest.value,
	greaterValue	:= greaterValue.value,
	message			:= ''
);

THIS^.AssertEquals_BOOL(
	Expected 	:= assertionIsWrong,
	Actual 		:= THIS^.assertorContainer.wasAssertionWrong,
	Message 	:= messageStringBuilder.sOut
);
END_METHOD

(*

short summary
==================
This test method tests ``assert.float.double.valueIsMax``
method of CNM_AssertionInterfaces library, 
it provides the possibility to handover test data via parameter 


.. <legal notes>

legal notes
=================
| SPDX-FileCopyrightText: © 2022 ekvip automation GmbH <info@ekvip.de>
| SPDX-License-Identifier: Apache-2.0
| For details check: Apache-2.0_

.. _Apache-2.0: https://www.apache.org/licenses/LICENSE-2.0

.. </legal notes>

parameters
==========

*)

METHOD testValueIsMax 
VAR_INPUT
	(* for the test it's the parameter ``currentValue`` *)
	valueToTest		:LRealTestParameter;
	(* for the test it's the parameter ``greaterValue`` *)
	maximumValue	:LRealTestParameter;
END_VAR
VAR
	(* just the expectation if the assertion to test must be worng or true *)
	assertionIsWrong		:BOOL;
	(* contains the format string for the test message *)
	message					:Tc2_System.T_MaxString;
	(* TwinCAT printf with the test message *)
	messageStringBuilder	:Tc2_Utilities.FB_FormatString;
	(* just to cast *)
	binaryCurrentValue		:POINTER TO LWORD;
	(* just to cast *)
	binaryMaximumValue		:POINTER TO LWORD;
	(* value of the paramter ``valueToTest`` as string *)
	valueToTestAsString		:Tc2_System.T_MaxString;
	(* value of the paramter ``maximumValue`` as string *)
	maximumValueAsString	:Tc2_System.T_MaxString;	
END_VAR
THIS^.assertorContainer.resetAssertor();

IF (
	Tc2_Utilities.LrealIsNaN(valueToTest.value)
	OR Tc2_Utilities.LrealIsNaN(maximumValue.value)
) THEN
	assertionIsWrong := TRUE;
ELSIF (
	(NOT Tc2_Utilities.LrealIsFinite(valueToTest.value))
	AND (NOT Tc2_Utilities.LrealIsFinite(maximumValue.value))
) THEN
	binaryCurrentValue := ADR(valueToTest.value);
	binaryMaximumValue := ADR(maximumValue.value);
	assertionIsWrong := (
		(NOT binaryCurrentValue^.SIGN) //inf
		AND (binaryMaximumValue^.SIGN) //-inf
	);
ELSIF (
	(NOT Tc2_Utilities.LrealIsFinite(valueToTest.value))
	AND (Tc2_Utilities.LrealIsFinite(maximumValue.value))
) THEN
	binaryCurrentValue := ADR(valueToTest.value);
	assertionIsWrong := (NOT binaryCurrentValue^.SIGN); //inf
ELSIF (
	(Tc2_Utilities.LrealIsFinite(valueToTest.value))
	AND (NOT Tc2_Utilities.LrealIsFinite(maximumValue.value))
) THEN
	binaryMaximumValue := ADR(maximumValue.value);
	assertionIsWrong := (binaryMaximumValue^.SIGN);//-inf
ELSE
	assertionIsWrong := (valueToTest.value > maximumValue.value);
END_IF

message := SEL(
	assertionIsWrong,
	'currentValue is %s maximumValue is %s assertion must be TRUE', 
	'currentValue is %s maximumValue is %s assertion must be FALSE'
);

valueToTestAsString := valueToTest.asString;
maximumValueAsString := maximumValue.asString;

messageStringBuilder(
	sFormat := message,
	arg1 := THIS^.AnyToArg(valueToTestAsString),
	arg2 := THIS^.AnyToArg(maximumValueAsString)
);

THIS^.assertorContainer.assertor.assert.float.double.valueIsMax(
	currentValue	:= valueToTest.value,
	maximumValue	:= maximumValue.value,
	message			:= ''
);

THIS^.AssertEquals_BOOL(
	Expected 	:= assertionIsWrong,
	Actual 		:= THIS^.assertorContainer.wasAssertionWrong,
	Message 	:= messageStringBuilder.sOut
);
END_METHOD

(*

short summary
==================
This test method tests ``assert.float.double.valueIsMin``
method of CNM_AssertionInterfaces library, 
it provides the possibility to handover test data via parameter 


.. <legal notes>

legal notes
=================
| SPDX-FileCopyrightText: © 2022 ekvip automation GmbH <info@ekvip.de>
| SPDX-License-Identifier: Apache-2.0
| For details check: Apache-2.0_

.. _Apache-2.0: https://www.apache.org/licenses/LICENSE-2.0

.. </legal notes>

parameters
==========

*)

METHOD testValueIsMin 
VAR_INPUT
	(* for the test it's the parameter ``currentValue`` *)
	valueToTest		:LRealTestParameter;
	(* for the test it's the parameter ``minimumValue`` *)
	minimumValue	:LRealTestParameter;
END_VAR
VAR
	(* just the expectation if the assertion to test must be worng or true *)
	assertionIsWrong		:BOOL;
	(* contains the format string for the test message *)
	message					:Tc2_System.T_MaxString;
	(* TwinCAT printf with the test message *)
	messageStringBuilder	:Tc2_Utilities.FB_FormatString;
	(* just to cast *)
	binaryCurrentValue		:POINTER TO LWORD;
	(* just to cast *)
	binaryMinimumValue		:POINTER TO LWORD;
	(* value of the paramter ``valueToTest`` as string *)
	valueToTestAsString		:Tc2_System.T_MaxString;
	(* value of the paramter ``minimumValue`` as string *)
	minimumValueAsString	:Tc2_System.T_MaxString;	
END_VAR
THIS^.assertorContainer.resetAssertor();

IF (
	Tc2_Utilities.LrealIsNaN(valueToTest.value)
	OR Tc2_Utilities.LrealIsNaN(minimumValue.value)
) THEN
	assertionIsWrong := TRUE;
ELSIF (
	(NOT Tc2_Utilities.LrealIsFinite(valueToTest.value))
	AND (NOT Tc2_Utilities.LrealIsFinite(minimumValue.value))
) THEN
	binaryCurrentValue := ADR(valueToTest.value);
	binaryMinimumValue := ADR(minimumValue.value);
	assertionIsWrong := (
		(binaryCurrentValue^.SIGN) //-inf
		AND (NOT binaryMinimumValue^.SIGN) //inf
	);
ELSIF (
	(NOT Tc2_Utilities.LrealIsFinite(valueToTest.value))
	AND (Tc2_Utilities.LrealIsFinite(minimumValue.value))
) THEN
	binaryCurrentValue := ADR(valueToTest.value);
	assertionIsWrong := (binaryCurrentValue^.SIGN);
ELSIF (
	(Tc2_Utilities.LrealIsFinite(valueToTest.value))
	AND (NOT Tc2_Utilities.LrealIsFinite(minimumValue.value))
) THEN
	binaryMinimumValue := ADR(minimumValue.value);
	assertionIsWrong := (NOT binaryMinimumValue^.SIGN);
ELSE
	assertionIsWrong := (valueToTest.value < minimumValue.value);
END_IF

message := SEL(
	assertionIsWrong,
	'currentValue is %s minimumValue is %s assertion must be TRUE', 
	'currentValue is %s minimumValue is %s assertion must be FALSE'
);

valueToTestAsString := valueToTest.asString;
minimumValueAsString := minimumValue.asString;

messageStringBuilder(
	sFormat := message,
	arg1 := THIS^.AnyToArg(valueToTestAsString),
	arg2 := THIS^.AnyToArg(minimumValueAsString)
);

THIS^.assertorContainer.assertor.assert.float.double.valueIsMin(
	currentValue	:= valueToTest.value,
	minimumValue	:= minimumValue.value,
	message			:= ''
);

THIS^.AssertEquals_BOOL(
	Expected 	:= assertionIsWrong,
	Actual 		:= THIS^.assertorContainer.wasAssertionWrong,
	Message 	:= messageStringBuilder.sOut
);
END_METHOD

(*

short summary
==================
This test method tests ``assert.float.double.valueIsNaN``
method of CNM_AssertionInterfaces library, 
it provides the possibility to handover test data via parameter 

.. <legal notes>

legal notes
=================
| SPDX-FileCopyrightText: © 2022 ekvip automation GmbH <info@ekvip.de>
| SPDX-License-Identifier: Apache-2.0
| For details check: Apache-2.0_

.. _Apache-2.0: https://www.apache.org/licenses/LICENSE-2.0

.. </legal notes>

parameters
==========

*)

METHOD testValueIsNaN
VAR_INPUT
	(* for the test it's the parameter ``currentValue`` *)
	valueToTest	:LRealTestParameter;	
END_VAR
VAR
	(* just the expectation if the assertion to test must be worng or true *)
	assertionIsWrong		:BOOL;
	(* contains the format string for the test message *)
	message					:Tc2_System.T_MaxString;
	(* TwinCAT printf with the test message *)
	messageStringBuilder	:Tc2_Utilities.FB_FormatString;
	(* value of the paramter ``valueToTest`` as string *)
	valueToTestAsString		:Tc2_System.T_MaxString;
END_VAR
THIS^.assertorContainer.resetAssertor();

assertionIsWrong := (NOT Tc2_Utilities.LrealIsNaN(valueToTest.value));

message := SEL(
	assertionIsWrong,
	'currentValue is %s assertion must be TRUE', 
	'currentValue is %s assertion must be FALSE'
);

valueToTestAsString := valueToTest.asString;

messageStringBuilder(
	sFormat := message,
	arg1 := THIS^.AnyToArg(valueToTestAsString)
);

THIS^.assertorContainer.assertor.assert.float.double.valueIsNaN(
	currentValue := valueToTest.value,
	message := ''
);

THIS^.AssertEquals_BOOL(
	Expected 	:= assertionIsWrong,
	Actual 		:= THIS^.assertorContainer.wasAssertionWrong,
	Message 	:= messageStringBuilder.sOut
);
END_METHOD

(*

short summary
==================
This test method tests ``assert.float.double.valueIsNegative``
method of CNM_AssertionInterfaces library, 
it provides the possibility to handover test data via parameter 

.. <legal notes>

legal notes
=================
| SPDX-FileCopyrightText: © 2022 ekvip automation GmbH <info@ekvip.de>
| SPDX-License-Identifier: Apache-2.0
| For details check: Apache-2.0_

.. _Apache-2.0: https://www.apache.org/licenses/LICENSE-2.0

.. </legal notes>

parameters
==========

*)

METHOD testValueIsNegative
VAR_INPUT
	(* for the test it's the parameter ``currentValue`` *)
	valueToTest	:LRealTestParameter;	
END_VAR
VAR
	(* just the expectation if the assertion to test must be worng or true *)
	assertionIsWrong		:BOOL;
	(* contains the format string for the test message *)
	message					:Tc2_System.T_MaxString;
	(* TwinCAT printf with the test message *)
	messageStringBuilder	:Tc2_Utilities.FB_FormatString;
	(* value of the paramter ``valueToTest`` as string *)
	valueToTestAsString		:Tc2_System.T_MaxString;
	(* binary value of the parameter ``valueToTest`` *)
	binaryValueToTest		:POINTER TO LWORD;
	(* sgin bit as BYTE for the message *)
	signBitAsByte			:BYTE;
	(* sgin bit as BOOL for the message *)
	signBit					:BOOL;	
END_VAR
THIS^.assertorContainer.resetAssertor();

binaryValueToTest := ADR(valueToTest.value);
signBit := binaryValueToTest^.SIGN;
signBitAsByte := TO_BYTE(signBit);
assertionIsWrong := (
	(NOT signBit)
	OR_ELSE Tc2_Utilities.LrealIsNaN(valueToTest.value)
);

message := SEL(
	assertionIsWrong,
	'currentValue is %s and sign bit is %u assertion must be TRUE', 
	'currentValue is %s and sign bit is %u assertion must be FALSE'
);

valueToTestAsString := valueToTest.asString;

messageStringBuilder(
	sFormat := message,
	arg1 := THIS^.AnyToArg(valueToTestAsString),
	arg2 := THIS^.AnyToArg(signBitAsByte)
);

THIS^.assertorContainer.assertor.assert.float.double.valueIsNegative(
	currentValue := valueToTest.value,
	message := ''
);

THIS^.AssertEquals_BOOL(
	Expected 	:= assertionIsWrong,
	Actual 		:= THIS^.assertorContainer.wasAssertionWrong,
	Message 	:= messageStringBuilder.sOut
);
END_METHOD

(*

short summary
==================
This test method tests ``assert.float.double.valueIsNegativeInfinite``
method of CNM_AssertionInterfaces library, 
it provides the possibility to handover test data via parameter 

.. <legal notes>

legal notes
=================
| SPDX-FileCopyrightText: © 2022 ekvip automation GmbH <info@ekvip.de>
| SPDX-License-Identifier: Apache-2.0
| For details check: Apache-2.0_

.. _Apache-2.0: https://www.apache.org/licenses/LICENSE-2.0

.. </legal notes>

parameters
==========

*)

METHOD testValueIsNegativeInfinite
VAR_INPUT
	(* for the test it's the parameter ``currentValue`` *)
	valueToTest	:LRealTestParameter;	
END_VAR
VAR
	(* just the expectation if the assertion to test must be worng or true *)
	assertionIsWrong		:BOOL;
	(* contains the format string for the test message *)
	message					:Tc2_System.T_MaxString;
	(* TwinCAT printf with the test message *)
	messageStringBuilder	:Tc2_Utilities.FB_FormatString;
	(* value of the paramter ``valueToTest`` as string *)
	valueToTestAsString		:Tc2_System.T_MaxString;
	(* binary value of the parameter ``valueToTest`` *)
	binaryValueToTest		:POINTER TO LWORD;
END_VAR
THIS^.assertorContainer.resetAssertor();

binaryValueToTest := ADR(valueToTest.value);
assertionIsWrong := (binaryValueToTest^ <> THIS^.BINARY_NEGATIVE_INFINITY);

message := SEL(
	assertionIsWrong,
	'currentValue is %s assertion must be TRUE', 
	'currentValue is %s assertion must be FALSE'
);

valueToTestAsString := valueToTest.asString;

messageStringBuilder(
	sFormat := message,
	arg1 := THIS^.AnyToArg(valueToTestAsString)
);

THIS^.assertorContainer.assertor.assert.float.double.valueIsNegativeInfinite(
	currentValue := valueToTest.value,
	message := ''
);

THIS^.AssertEquals_BOOL(
	Expected 	:= assertionIsWrong,
	Actual 		:= THIS^.assertorContainer.wasAssertionWrong,
	Message 	:= messageStringBuilder.sOut
);
END_METHOD

(*

short summary
==================
This test method tests ``assert.float.double.valueIsNegativeZero``
method of CNM_AssertionInterfaces library, 
it provides the possibility to handover test data via parameter 

.. <legal notes>

legal notes
=================
| SPDX-FileCopyrightText: © 2022 ekvip automation GmbH <info@ekvip.de>
| SPDX-License-Identifier: Apache-2.0
| For details check: Apache-2.0_

.. _Apache-2.0: https://www.apache.org/licenses/LICENSE-2.0

.. </legal notes>

parameters
==========

*)

METHOD testValueIsNegativeZero
VAR_INPUT
	(* for the test it's the parameter ``currentValue`` *)
	valueToTest	:LRealTestParameter;	
END_VAR
VAR
	(* just the expectation if the assertion to test must be worng or true *)
	assertionIsWrong		:BOOL;
	(* contains the format string for the test message *)
	message					:Tc2_System.T_MaxString;
	(* TwinCAT printf with the test message *)
	messageStringBuilder	:Tc2_Utilities.FB_FormatString;
	(* value of the paramter ``valueToTest`` as string *)
	valueToTestAsString		:Tc2_System.T_MaxString;
	(* binary value of the parameter ``valueToTest`` *)
	binaryValueToTest		:POINTER TO LWORD;
	(* sgin bit as BYTE for the message *)
	signBitAsByte			:BYTE;
	(* sgin bit as BOOL for the message *)
	signBit					:BOOL;	
END_VAR
THIS^.assertorContainer.resetAssertor();

binaryValueToTest := ADR(valueToTest.value);
signBit := binaryValueToTest^.SIGN;
signBitAsByte := TO_BYTE(signBit);

assertionIsWrong := (binaryValueToTest^ <> THIS^.BINARY_MINUS_ZERO);

message := SEL(
	assertionIsWrong,
	'currentValue is %s and sign bit is %u assertion must be TRUE', 
	'currentValue is %s and sign bit is %u assertion must be FALSE'
);

valueToTestAsString := valueToTest.asString;

messageStringBuilder(
	sFormat := message,
	arg1 := THIS^.AnyToArg(valueToTestAsString),
	arg2 := THIS^.AnyToArg(signBitAsByte)
);

THIS^.assertorContainer.assertor.assert.float.double.valueIsNegativeZero(
	currentValue := valueToTest.value,
	message := ''
);

THIS^.AssertEquals_BOOL(
	Expected 	:= assertionIsWrong,
	Actual 		:= THIS^.assertorContainer.wasAssertionWrong,
	Message 	:= messageStringBuilder.sOut
);
END_METHOD

(*

short summary
==================
This test method tests ``assert.float.double.valueIsNormal``
method of CNM_AssertionInterfaces library, 
it provides the possibility to handover test data via parameter 

.. <legal notes>

legal notes
=================
| SPDX-FileCopyrightText: © 2022 ekvip automation GmbH <info@ekvip.de>
| SPDX-License-Identifier: Apache-2.0
| For details check: Apache-2.0_

.. _Apache-2.0: https://www.apache.org/licenses/LICENSE-2.0

.. </legal notes>

parameters
==========

*)

METHOD testValueIsNormal
VAR_INPUT
	(* for the test it's the parameter ``currentValue`` *)
	valueToTest	:LRealTestParameter;	
END_VAR
VAR
	(* just the expectation if the assertion to test must be worng or true *)
	assertionIsWrong		:BOOL;
	(* contains the format string for the test message *)
	message					:Tc2_System.T_MaxString;
	(* TwinCAT printf with the test message *)
	messageStringBuilder	:Tc2_Utilities.FB_FormatString;
	(* value of the paramter ``valueToTest`` as string *)
	valueToTestAsString		:Tc2_System.T_MaxString;
	(* binary value of the parameter ``valueToTest`` *)
	binaryValueToTest		:POINTER TO LWORD;
END_VAR
THIS^.assertorContainer.resetAssertor();

binaryValueToTest := ADR(valueToTest.value);

assertionIsWrong := (
	((binaryValueToTest^ AND THIS^.MASK_FOR_EXPONENT) = THIS^.BINARY_ZERO)
	OR_ELSE Tc2_Utilities.LrealIsNaN(valueToTest.value)
	OR_ELSE (NOT Tc2_Utilities.LrealIsFinite(valueToTest.value))
);

message := SEL(
	assertionIsWrong,
	'currentValue is %s assertion must be TRUE', 
	'currentValue is %s assertion must be FALSE'
);

valueToTestAsString := valueToTest.asString;

messageStringBuilder(
	sFormat := message,
	arg1 := THIS^.AnyToArg(valueToTestAsString)
);

THIS^.assertorContainer.assertor.assert.float.double.valueIsNormal(
	currentValue := valueToTest.value,
	message := ''
);

THIS^.AssertEquals_BOOL(
	Expected 	:= assertionIsWrong,
	Actual 		:= THIS^.assertorContainer.wasAssertionWrong,
	Message 	:= messageStringBuilder.sOut
);
END_METHOD

(*

short summary
==================
This test method tests ``assert.float.double.valueIsNotEqualTo``
method of CNM_AssertionInterfaces library, 
it provides the possibility to handover test data via parameter 


.. <legal notes>

legal notes
=================
| SPDX-FileCopyrightText: © 2022 ekvip automation GmbH <info@ekvip.de>
| SPDX-License-Identifier: Apache-2.0
| For details check: Apache-2.0_

.. _Apache-2.0: https://www.apache.org/licenses/LICENSE-2.0

.. </legal notes>

parameters
==========

*)

METHOD testValueIsNotEqualTo 
VAR_INPUT
	(* for the test it's the parameter ``currentValue`` *)
	valueToTest		:LRealTestParameter;
	(* for the test it's the parameter ``unexpectedValue`` *)
	unexpectedValue	:LRealTestParameter;
	(* for the test it's the parameter ``tolerance`` *)
	tolerance		:LRealTestParameter;
END_VAR
VAR
	(* just the expectation if the assertion to test must be worng or true *)
	assertionIsWrong		:BOOL;
	(* contains the format string for the test message *)
	message					:Tc2_System.T_MaxString;
	(* TwinCAT printf with the test message *)
	messageStringBuilder	:Tc2_Utilities.FB_FormatString;
	(* just to cast *)
	binaryCurrentValue		:POINTER TO LWORD;
	(* just to cast *)
	binaryUnexpectedValue	:POINTER TO LWORD;
	(* value of the paramter ``valueToTest`` as string *)
	valueToTestAsString		:Tc2_System.T_MaxString;
	(* value of the paramter ``unexpectedValue`` as string *)
	unexpectedValueAsString	:Tc2_System.T_MaxString;
	(* value of the paramter ``tolerance`` as string *)
	toleranceAsString		:Tc2_System.T_MaxString;	
END_VAR
THIS^.assertorContainer.resetAssertor();
IF (
	Tc2_Utilities.LrealIsNaN(valueToTest.value)
	OR Tc2_Utilities.LrealIsNaN(unexpectedValue.value)
	OR Tc2_Utilities.LrealIsNaN(tolerance.value)
) THEN
	assertionIsWrong := FALSE;
ELSIF (NOT Tc2_Utilities.LrealIsFinite(tolerance.value)) THEN
	assertionIsWrong := TRUE;
ELSIF (
	Tc2_Utilities.LrealIsFinite(valueToTest.value)
	<> Tc2_Utilities.LrealIsFinite(unexpectedValue.value)
) THEN
	assertionIsWrong := FALSE; 
ELSIF (
	(NOT Tc2_Utilities.LrealIsFinite(valueToTest.value))
	OR (NOT Tc2_Utilities.LrealIsFinite(unexpectedValue.value))
) THEN
	binaryCurrentValue := ADR(valueToTest.value);
	binaryUnexpectedValue := ADR(unexpectedValue.value);
	assertionIsWrong := (binaryCurrentValue^.SIGN = binaryUnexpectedValue^.SIGN);
ELSE
	assertionIsWrong := (
		((unexpectedValue.value + ABS(tolerance.value)) >= valueToTest.value)
		AND ((unexpectedValue.value - ABS(tolerance.value)) <= valueToTest.value)
	);
END_IF

message := SEL(
	assertionIsWrong,
	'currentValue is %s unexpectedValue is %s tolerance is %s assertion must be TRUE', 
	'currentValue is %s unexpectedValue is %s tolerance is %s assertion must be FALSE'
);

valueToTestAsString := valueToTest.asString;
unexpectedValueAsString := unexpectedValue.asString;
toleranceAsString := tolerance.asString;

messageStringBuilder(
	sFormat := message,
	arg1 := THIS^.AnyToArg(valueToTestAsString),
	arg2 := THIS^.AnyToArg(unexpectedValueAsString),
	arg3 := THIS^.AnyToArg(toleranceAsString)
);

THIS^.assertorContainer.assertor.assert.float.double.valueIsNotEqualTo(
	currentValue	:= valueToTest.value,
	unexpectedValue	:= unexpectedValue.value,
	tolerance       := tolerance.value,
	message			:= ''
);

THIS^.AssertEquals_BOOL(
	Expected 	:= assertionIsWrong,
	Actual 		:= THIS^.assertorContainer.wasAssertionWrong,
	Message 	:= messageStringBuilder.sOut
);
END_METHOD

(*

short summary
==================
This test method tests ``assert.float.double.valueIsNotNegativeInfinite``
method of CNM_AssertionInterfaces library, 
it provides the possibility to handover test data via parameter 

.. <legal notes>

legal notes
=================
| SPDX-FileCopyrightText: © 2022 ekvip automation GmbH <info@ekvip.de>
| SPDX-License-Identifier: Apache-2.0
| For details check: Apache-2.0_

.. _Apache-2.0: https://www.apache.org/licenses/LICENSE-2.0

.. </legal notes>

parameters
==========

*)

METHOD testValueIsNotNegativeInfinite
VAR_INPUT
	(* for the test it's the parameter ``currentValue`` *)
	valueToTest	:LRealTestParameter;	
END_VAR
VAR
	(* just the expectation if the assertion to test must be worng or true *)
	assertionIsWrong		:BOOL;
	(* contains the format string for the test message *)
	message					:Tc2_System.T_MaxString;
	(* TwinCAT printf with the test message *)
	messageStringBuilder	:Tc2_Utilities.FB_FormatString;
	(* value of the paramter ``valueToTest`` as string *)
	valueToTestAsString		:Tc2_System.T_MaxString;
	(* binary value of the parameter ``valueToTest`` *)
	binaryValueToTest		:POINTER TO LWORD;
END_VAR
THIS^.assertorContainer.resetAssertor();

binaryValueToTest := ADR(valueToTest.value);
assertionIsWrong := (binaryValueToTest^ = THIS^.BINARY_NEGATIVE_INFINITY);

message := SEL(
	assertionIsWrong,
	'currentValue is %s assertion must be TRUE', 
	'currentValue is %s assertion must be FALSE'
);

valueToTestAsString := valueToTest.asString;

messageStringBuilder(
	sFormat := message,
	arg1 := THIS^.AnyToArg(valueToTestAsString)
);

THIS^.assertorContainer.assertor.assert.float.double.valueIsNotNegativeInfinite(
	currentValue := valueToTest.value,
	message := ''
);

THIS^.AssertEquals_BOOL(
	Expected 	:= assertionIsWrong,
	Actual 		:= THIS^.assertorContainer.wasAssertionWrong,
	Message 	:= messageStringBuilder.sOut
);
END_METHOD

(*

short summary
==================
This test method tests ``assert.float.double.valueIsNotPositiveInfinite``
method of CNM_AssertionInterfaces library, 
it provides the possibility to handover test data via parameter 

.. <legal notes>

legal notes
=================
| SPDX-FileCopyrightText: © 2022 ekvip automation GmbH <info@ekvip.de>
| SPDX-License-Identifier: Apache-2.0
| For details check: Apache-2.0_

.. _Apache-2.0: https://www.apache.org/licenses/LICENSE-2.0

.. </legal notes>

parameters
==========

*)

METHOD testValueIsNotPositiveInfinite
VAR_INPUT
	(* for the test it's the parameter ``currentValue`` *)
	valueToTest	:LRealTestParameter;	
END_VAR
VAR
	(* just the expectation if the assertion to test must be worng or true *)
	assertionIsWrong		:BOOL;
	(* contains the format string for the test message *)
	message					:Tc2_System.T_MaxString;
	(* TwinCAT printf with the test message *)
	messageStringBuilder	:Tc2_Utilities.FB_FormatString;
	(* value of the paramter ``valueToTest`` as string *)
	valueToTestAsString		:Tc2_System.T_MaxString;
	(* binary value of the parameter ``valueToTest`` *)
	binaryValueToTest		:POINTER TO LWORD;
END_VAR
THIS^.assertorContainer.resetAssertor();

binaryValueToTest := ADR(valueToTest.value);
assertionIsWrong := (binaryValueToTest^ = THIS^.BINARY_INFINITY);

message := SEL(
	assertionIsWrong,
	'currentValue is %s assertion must be TRUE', 
	'currentValue is %s assertion must be FALSE'
);

valueToTestAsString := valueToTest.asString;

messageStringBuilder(
	sFormat := message,
	arg1 := THIS^.AnyToArg(valueToTestAsString)
);

THIS^.assertorContainer.assertor.assert.float.double.valueIsNotPositiveInfinite(
	currentValue := valueToTest.value,
	message := ''
);

THIS^.AssertEquals_BOOL(
	Expected 	:= assertionIsWrong,
	Actual 		:= THIS^.assertorContainer.wasAssertionWrong,
	Message 	:= messageStringBuilder.sOut
);
END_METHOD

(*

short summary
==================
This test method tests ``assert.float.double.valueIsNotSpecial``
method of CNM_AssertionInterfaces library, 
it provides the possibility to handover test data via parameter 

.. <legal notes>

legal notes
=================
| SPDX-FileCopyrightText: © 2022 ekvip automation GmbH <info@ekvip.de>
| SPDX-License-Identifier: Apache-2.0
| For details check: Apache-2.0_

.. _Apache-2.0: https://www.apache.org/licenses/LICENSE-2.0

.. </legal notes>

parameters
==========

*)

METHOD testValueIsNotSpecial
VAR_INPUT
	(* for the test it's the parameter ``currentValue`` *)
	valueToTest	:LRealTestParameter;	
END_VAR
VAR
	(* just the expectation if the assertion to test must be worng or true *)
	assertionIsWrong		:BOOL;
	(* contains the format string for the test message *)
	message					:Tc2_System.T_MaxString;
	(* TwinCAT printf with the test message *)
	messageStringBuilder	:Tc2_Utilities.FB_FormatString;
	(* value of the paramter ``valueToTest`` as string *)
	valueToTestAsString		:Tc2_System.T_MaxString;
END_VAR
THIS^.assertorContainer.resetAssertor();

assertionIsWrong := (
	(NOT Tc2_Utilities.LrealIsFinite(valueToTest.value))
	OR_ELSE Tc2_Utilities.LrealIsNaN(valueToTest.value)
);

message := SEL(
	assertionIsWrong,
	'currentValue is %s assertion must be TRUE', 
	'currentValue is %s assertion must be FALSE'
);

valueToTestAsString := valueToTest.asString;

messageStringBuilder(
	sFormat := message,
	arg1 := THIS^.AnyToArg(valueToTestAsString)
);

THIS^.assertorContainer.assertor.assert.float.double.valueIsNotSpecial(
	currentValue := valueToTest.value,
	message := ''
);

THIS^.AssertEquals_BOOL(
	Expected 	:= assertionIsWrong,
	Actual 		:= THIS^.assertorContainer.wasAssertionWrong,
	Message 	:= messageStringBuilder.sOut
);
END_METHOD

(*

short summary
==================
This test method tests ``assert.float.double.valueIsPositive``
method of CNM_AssertionInterfaces library, 
it provides the possibility to handover test data via parameter 

.. <legal notes>

legal notes
=================
| SPDX-FileCopyrightText: © 2022 ekvip automation GmbH <info@ekvip.de>
| SPDX-License-Identifier: Apache-2.0
| For details check: Apache-2.0_

.. _Apache-2.0: https://www.apache.org/licenses/LICENSE-2.0

.. </legal notes>

parameters
==========

*)

METHOD testValueIsPositive
VAR_INPUT
	(* for the test it's the parameter ``currentValue`` *)
	valueToTest	:LRealTestParameter;	
END_VAR
VAR
	(* just the expectation if the assertion to test must be worng or true *)
	assertionIsWrong		:BOOL;
	(* contains the format string for the test message *)
	message					:Tc2_System.T_MaxString;
	(* TwinCAT printf with the test message *)
	messageStringBuilder	:Tc2_Utilities.FB_FormatString;
	(* value of the paramter ``valueToTest`` as string *)
	valueToTestAsString		:Tc2_System.T_MaxString;
	(* binary value of the parameter ``valueToTest`` *)
	binaryValueToTest		:POINTER TO LWORD;
	(* sgin bit as BYTE for the message *)
	signBitAsByte			:BYTE;
	(* sgin bit as BOOL for the message *)
	signBit					:BOOL;	
END_VAR
THIS^.assertorContainer.resetAssertor();

binaryValueToTest := ADR(valueToTest.value);
signBit := binaryValueToTest^.SIGN;
signBitAsByte := TO_BYTE(signBit);
assertionIsWrong := (
	signBit
	OR Tc2_Utilities.LrealIsNaN(valueToTest.value)
);

message := SEL(
	assertionIsWrong,
	'currentValue is %s and sign bit is %u assertion must be TRUE', 
	'currentValue is %s and sign bit is %u assertion must be FALSE'
);

valueToTestAsString := valueToTest.asString;

messageStringBuilder(
	sFormat := message,
	arg1 := THIS^.AnyToArg(valueToTestAsString),
	arg2 := THIS^.AnyToArg(signBitAsByte)
);

THIS^.assertorContainer.assertor.assert.float.double.valueIsPositive(
	currentValue := valueToTest.value,
	message := ''
);

THIS^.AssertEquals_BOOL(
	Expected 	:= assertionIsWrong,
	Actual 		:= THIS^.assertorContainer.wasAssertionWrong,
	Message 	:= messageStringBuilder.sOut
);
END_METHOD

(*

short summary
==================
This test method tests ``assert.float.double.valueIsPositiveInfinite``
method of CNM_AssertionInterfaces library, 
it provides the possibility to handover test data via parameter 

.. <legal notes>

legal notes
=================
| SPDX-FileCopyrightText: © 2022 ekvip automation GmbH <info@ekvip.de>
| SPDX-License-Identifier: Apache-2.0
| For details check: Apache-2.0_

.. _Apache-2.0: https://www.apache.org/licenses/LICENSE-2.0

.. </legal notes>

parameters
==========

*)

METHOD testValueIsPositiveInfinite
VAR_INPUT
	(* for the test it's the parameter ``currentValue`` *)
	valueToTest	:LRealTestParameter;	
END_VAR
VAR
	(* just the expectation if the assertion to test must be worng or true *)
	assertionIsWrong		:BOOL;
	(* contains the format string for the test message *)
	message					:Tc2_System.T_MaxString;
	(* TwinCAT printf with the test message *)
	messageStringBuilder	:Tc2_Utilities.FB_FormatString;
	(* value of the paramter ``valueToTest`` as string *)
	valueToTestAsString		:Tc2_System.T_MaxString;
	(* binary value of the parameter ``valueToTest`` *)
	binaryValueToTest		:POINTER TO LWORD;
END_VAR
THIS^.assertorContainer.resetAssertor();

binaryValueToTest := ADR(valueToTest.value);
assertionIsWrong := (binaryValueToTest^ <> THIS^.BINARY_INFINITY);

message := SEL(
	assertionIsWrong,
	'currentValue is %s assertion must be TRUE', 
	'currentValue is %s assertion must be FALSE'
);

valueToTestAsString := valueToTest.asString;

messageStringBuilder(
	sFormat := message,
	arg1 := THIS^.AnyToArg(valueToTestAsString)
);

THIS^.assertorContainer.assertor.assert.float.double.valueIsPositiveInfinite(
	currentValue := valueToTest.value,
	message := ''
);

THIS^.AssertEquals_BOOL(
	Expected 	:= assertionIsWrong,
	Actual 		:= THIS^.assertorContainer.wasAssertionWrong,
	Message 	:= messageStringBuilder.sOut
);
END_METHOD

(*

short summary
==================
This test method tests ``assert.float.double.valueIsPositiveZero``
method of CNM_AssertionInterfaces library, 
it provides the possibility to handover test data via parameter 

.. <legal notes>

legal notes
=================
| SPDX-FileCopyrightText: © 2022 ekvip automation GmbH <info@ekvip.de>
| SPDX-License-Identifier: Apache-2.0
| For details check: Apache-2.0_

.. _Apache-2.0: https://www.apache.org/licenses/LICENSE-2.0

.. </legal notes>

parameters
==========

*)

METHOD testValueIsPositiveZero
VAR_INPUT
	(* for the test it's the parameter ``currentValue`` *)
	valueToTest	:LRealTestParameter;	
END_VAR
VAR
	(* just the expectation if the assertion to test must be worng or true *)
	assertionIsWrong		:BOOL;
	(* contains the format string for the test message *)
	message					:Tc2_System.T_MaxString;
	(* TwinCAT printf with the test message *)
	messageStringBuilder	:Tc2_Utilities.FB_FormatString;
	(* value of the paramter ``valueToTest`` as string *)
	valueToTestAsString		:Tc2_System.T_MaxString;
	(* binary value of the parameter ``valueToTest`` *)
	binaryValueToTest		:POINTER TO LWORD;
	(* sgin bit as BYTE for the message *)
	signBitAsByte			:BYTE;
	(* sgin bit as BOOL for the message *)
	signBit					:BOOL;	
END_VAR
THIS^.assertorContainer.resetAssertor();

binaryValueToTest := ADR(valueToTest.value);
signBit := binaryValueToTest^.SIGN;
signBitAsByte := TO_BYTE(signBit);

assertionIsWrong := (binaryValueToTest^ <> THIS^.BINARY_ZERO);

message := SEL(
	assertionIsWrong,
	'currentValue is %s and sign bit is %u assertion must be TRUE', 
	'currentValue is %s and sign bit is %u assertion must be FALSE'
);

valueToTestAsString := valueToTest.asString;

messageStringBuilder(
	sFormat := message,
	arg1 := THIS^.AnyToArg(valueToTestAsString),
	arg2 := THIS^.AnyToArg(signBitAsByte)
);

THIS^.assertorContainer.assertor.assert.float.double.valueIsPositiveZero(
	currentValue := valueToTest.value,
	message := ''
);

THIS^.AssertEquals_BOOL(
	Expected 	:= assertionIsWrong,
	Actual 		:= THIS^.assertorContainer.wasAssertionWrong,
	Message 	:= messageStringBuilder.sOut
);
END_METHOD

(*

short summary
==================
This test method tests ``assert.float.double.valueIsSpecial``
method of CNM_AssertionInterfaces library, 
it provides the possibility to handover test data via parameter 

.. <legal notes>

legal notes
=================
| SPDX-FileCopyrightText: © 2022 ekvip automation GmbH <info@ekvip.de>
| SPDX-License-Identifier: Apache-2.0
| For details check: Apache-2.0_

.. _Apache-2.0: https://www.apache.org/licenses/LICENSE-2.0

.. </legal notes>

parameters
==========

*)

METHOD testValueIsSpecial
VAR_INPUT
	(* for the test it's the parameter ``currentValue`` *)
	valueToTest	:LRealTestParameter;	
END_VAR
VAR
	(* just the expectation if the assertion to test must be worng or true *)
	assertionIsWrong		:BOOL;
	(* contains the format string for the test message *)
	message					:Tc2_System.T_MaxString;
	(* TwinCAT printf with the test message *)
	messageStringBuilder	:Tc2_Utilities.FB_FormatString;
	(* value of the paramter ``valueToTest`` as string *)
	valueToTestAsString		:Tc2_System.T_MaxString;
END_VAR
THIS^.assertorContainer.resetAssertor();

assertionIsWrong := (
	(NOT Tc2_Utilities.LrealIsNaN(valueToTest.value))
	AND_THEN (Tc2_Utilities.LrealIsFinite(valueToTest.value))
);

message := SEL(
	assertionIsWrong,
	'currentValue is %s assertion must be TRUE', 
	'currentValue is %s assertion must be FALSE'
);

valueToTestAsString := valueToTest.asString;

messageStringBuilder(
	sFormat := message,
	arg1 := THIS^.AnyToArg(valueToTestAsString)
);

THIS^.assertorContainer.assertor.assert.float.double.valueIsSpecial(
	currentValue := valueToTest.value,
	message := ''
);

THIS^.AssertEquals_BOOL(
	Expected 	:= assertionIsWrong,
	Actual 		:= THIS^.assertorContainer.wasAssertionWrong,
	Message 	:= messageStringBuilder.sOut
);
END_METHOD

(*

short summary
==================
This test method tests ``assert.float.double.valueIsSubnormal``
method of CNM_AssertionInterfaces library, 
it provides the possibility to handover test data via parameter 

.. <legal notes>

legal notes
=================
| SPDX-FileCopyrightText: © 2022 ekvip automation GmbH <info@ekvip.de>
| SPDX-License-Identifier: Apache-2.0
| For details check: Apache-2.0_

.. _Apache-2.0: https://www.apache.org/licenses/LICENSE-2.0

.. </legal notes>

parameters
==========

*)

METHOD testValueIsSubnormal
VAR_INPUT
	(* for the test it's the parameter ``currentValue`` *)
	valueToTest	:LRealTestParameter;	
END_VAR
VAR
	(* just the expectation if the assertion to test must be worng or true *)
	assertionIsWrong		:BOOL;
	(* contains the format string for the test message *)
	message					:Tc2_System.T_MaxString;
	(* TwinCAT printf with the test message *)
	messageStringBuilder	:Tc2_Utilities.FB_FormatString;
	(* value of the paramter ``valueToTest`` as string *)
	valueToTestAsString		:Tc2_System.T_MaxString;
	(* binary value of the parameter ``valueToTest`` *)
	binaryValueToTest		:POINTER TO LWORD;
END_VAR
THIS^.assertorContainer.resetAssertor();

binaryValueToTest := ADR(valueToTest.value);

assertionIsWrong := (
	((binaryValueToTest^ AND THIS^.MASK_FOR_EXPONENT) <> THIS^.BINARY_ZERO)
);

message := SEL(
	assertionIsWrong,
	'currentValue is %s assertion must be TRUE', 
	'currentValue is %s assertion must be FALSE'
);

valueToTestAsString := valueToTest.asString;

messageStringBuilder(
	sFormat := message,
	arg1 := THIS^.AnyToArg(valueToTestAsString)
);

THIS^.assertorContainer.assertor.assert.float.double.valueIsSubnormal(
	currentValue := valueToTest.value,
	message := ''
);

THIS^.AssertEquals_BOOL(
	Expected 	:= assertionIsWrong,
	Actual 		:= THIS^.assertorContainer.wasAssertionWrong,
	Message 	:= messageStringBuilder.sOut
);
END_METHOD

END_FUNCTION_BLOCK

// ---- AssertionTester/AssertionTests/FloatAssertions/classes/RealAssertionTests.TcPOU
(*

short summary
==================
This class tests all methods of REAL assertions
with various combinations of inputs and checks expected 
outputs are satisfied or not

.. <legal notes>

legal notes
=================
| SPDX-FileCopyrightText: © 2022 ekvip automation GmbH <info@ekvip.de>
| SPDX-License-Identifier: Apache-2.0
| For details check: Apache-2.0_

.. _Apache-2.0: https://www.apache.org/licenses/LICENSE-2.0

.. </legal notes>

methods and properties
======================

*)


FUNCTION_BLOCK RealAssertionTests EXTENDS AbstractAssertorTest
VAR
	(* not a number *)
	NAN							:REAL;
	(* infinity *)
	INF							:REAL;
	(* -infinity *)
	MINUS_INF					:REAL;
	(* -0.0 (MSB is set only) *)
	MINUS_ZERO					:REAL;
	(* minimum subnormal value (all fraction bits and MSB set only) *)
	MIN_SUBNORMAL				:REAL;
	(* maximum subnormal value (all fraction bits are set only) *)
	MAX_SUBNORMAL				:REAL;
	(* smallest positive subnormal value (LSB set only)*)
	SMALLEST_POSITIVE_SUBNORMAL	:REAL;
	(* smallest negative subnormal value (LSB and MSB set only)*)
	SMALLEST_NEGATIVE_SUBNORMAL	:REAL;
END_VAR
VAR CONSTANT
	(* prefix to unify the test names *)
	TEST_NAME_PREFIX					:STRING := 'assert.float.single.';
	(* max value of real *)
	MAX_NON_SPECIAL						:REAL := 3.402823E+38;
	(* min value of real *)
	MIN_NON_SPECIAL						:REAL := -3.402823E+38;
	(* 0.0 *)
	ZERO								:REAL := 0.0;
	(* 1% *)
	ONE_PERCENT							:REAL := 0.01;
	(* 1‰ *)
	ONE_PERMILLE						:REAL := 0.001;
	(* bit number of the sign bit *)
	SIGN								:USINT := 31;
	(* binary value of 0.0 *)
	BINARY_ZERO							:DWORD := 16#0000_0000;
	(* binary value of -0.0 *)
	BINARY_MINUS_ZERO					:DWORD := 16#8000_0000;
	(* binary value of inf *)
	BINARY_INFINITY						:DWORD := 16#7F80_0000;
	(* binary value of -inf *)
	BINARY_NEGATIVE_INFINITY			:DWORD := 16#FF80_0000;
	(* mask to filter the exponent of the number *)
	MASK_FOR_EXPONENT					:DWORD := 16#7F80_0000;
	(* minimum denormalized number *)
	BINARY_MIN_SUBNORMAL				:DWORD := 16#807F_FFFF;
	(* maximum denormalized number*)
	BINARY_MAX_SUBNORMAL				:DWORD := 16#007F_FFFF;
	(* smallest positive denormalizied number greater than zero *)
	BINARY_SMALLEST_POSITIVE_SUBNORMAL	:DWORD := 16#0000_0001;
	(* smallest negative denormalizied number greater than minus zero *)
	BINARY_SMALLEST_NEGATIVE_SUBNORMAL	:DWORD := 16#8000_0001;
	(* smallest positive signaling NaN *)
	BINARY_POSITIVE_SIGNALING_NAN		:DWORD := 16#7F80_0001;
END_VAR

THIS^.runValueIsEqualToTests();
THIS^.runValueIsGreaterThanTests();
THIS^.runValueIsInRangeOfTests();
THIS^.runValueIsLessThanTests();
THIS^.runValueIsMaxTests();
THIS^.runValueIsMinTests();
THIS^.runValueIsNotEqualToTests();
THIS^.runValueIsANumberTests();
THIS^.runValueIsFiniteTests();
THIS^.runValueIsInfiniteTests();
THIS^.runValueIsNaNTests();
THIS^.runValueIsNegativeTests();
THIS^.runValueIsPositiveTests();
THIS^.runValueIsNegativeInfiniteTests();
THIS^.runValueIsPositiveInfiniteTests();
THIS^.runValueIsNegativeZeroTests();
THIS^.runValueIsPositiveZeroTests();
THIS^.runValueIsNormalTests();
THIS^.runValueIsNotNegativeInfiniteTests();
THIS^.runValueIsNotPositiveInfiniteTests();
THIS^.runValueIsNotSpecialTests();
THIS^.runValueIsSpecialTests();
THIS^.runValueIsSubnormalTests();

(*

short summary
=============
It attaches the container with the class to test
and it sets the special numbers from `IEEE 754`_ standard

.. _IEEE 754: https://en.wikipedia.org/wiki/IEEE_754

legal notes
=================
| SPDX-FileCopyrightText: © 2023 ekvip automation GmbH <info@ekvip.de>
| SPDX-License-Identifier: Apache-2.0
| For details check: Apache-2.0_

.. _Apache-2.0: https://www.apache.org/licenses/LICENSE-2.0

.. </legal notes>

parameters
==========

*)

METHOD FB_init :BOOL
VAR_INPUT
	(* if TRUE, the retain variables are initialized (warm start / cold start) *)
    bInitRetains	:BOOL;
	(* if TRUE, the instance afterwards gets moved into the copy code (online change) *)
    bInCopyCode		:BOOL;
	(* container with the class to test *)
	classToBeTested :IAssertorContainer;
END_VAR
VAR
	{attribute 'hide'}
	newHashstate3		:CNM_AbstractObject.Hashcode;
	{attribute 'hide'}
	binaryNumberPointer	:POINTER TO DWORD;	
END_VAR
VAR CONSTANT
	{attribute 'hide'}
	NUMBER_OF_LEFT_SHIFTS		:UINT	:= 17;
	{attribute 'hide'}
	NUMBER_OF_LEFT_ROTATIONS	:UINT   := 45;
END_VAR
binaryNumberPointer := ADR(THIS^.NAN);
binaryNumberPointer^ := THIS^.BINARY_POSITIVE_SIGNALING_NAN;

binaryNumberPointer := ADR(THIS^.INF);
binaryNumberPointer^ := THIS^.BINARY_INFINITY;

binaryNumberPointer := ADR(THIS^.MINUS_INF);
binaryNumberPointer^ := THIS^.BINARY_NEGATIVE_INFINITY;

binaryNumberPointer := ADR(THIS^.MINUS_ZERO);
binaryNumberPointer^ := THIS^.BINARY_MINUS_ZERO;

binaryNumberPointer := ADR(THIS^.MIN_SUBNORMAL);
binaryNumberPointer^ := THIS^.BINARY_MIN_SUBNORMAL; 

binaryNumberPointer := ADR(THIS^.MAX_SUBNORMAL);
binaryNumberPointer^ := THIS^.BINARY_MAX_SUBNORMAL; 

binaryNumberPointer := ADR(THIS^.SMALLEST_POSITIVE_SUBNORMAL);
binaryNumberPointer^ := THIS^.BINARY_SMALLEST_POSITIVE_SUBNORMAL; 

binaryNumberPointer := ADR(THIS^.SMALLEST_NEGATIVE_SUBNORMAL);
binaryNumberPointer^ := THIS^.BINARY_SMALLEST_NEGATIVE_SUBNORMAL;
END_METHOD

(*

short summary
==================
This test method is a helper function to create a unified test name

.. <legal notes>

legal notes
=================
| SPDX-FileCopyrightText: © 2022 ekvip automation GmbH <info@ekvip.de>
| SPDX-License-Identifier: Apache-2.0
| For details check: Apache-2.0_

.. _Apache-2.0: https://www.apache.org/licenses/LICENSE-2.0

.. </legal notes>

parameters
==========

*)

METHOD PROTECTED getTestNameFor :Tc2_System.T_MaxString
VAR_INPUT
	(* name of the method to test, to create a unified test name *)
	nameOfMethodToTest	:Tc2_System.T_MaxString;
END_VAR
getTestNameFor := Tc2_Standard.CONCAT(THIS^.TEST_NAME_PREFIX, nameOfMethodToTest);
END_METHOD

(*

short summary
==================
This test method tests ``assert.float.single.valueIsANumber``
method of CNM_AssertionInterfaces library with various inputs

.. <legal notes>

legal notes
=================
| SPDX-FileCopyrightText: © 2022 ekvip automation GmbH <info@ekvip.de>
| SPDX-License-Identifier: Apache-2.0
| For details check: Apache-2.0_

.. _Apache-2.0: https://www.apache.org/licenses/LICENSE-2.0

.. </legal notes>

*)

METHOD runValueIsANumberTests
RETURN (NOT TcUnit.TEST_ORDERED(THIS^.getTestNameFor('valueIsANumber')));

THIS^.testValueIsANumber(THIS^.NAN);
THIS^.testValueIsANumber(THIS^.INF);
THIS^.testValueIsANumber(THIS^.MINUS_INF);
THIS^.testValueIsANumber(THIS^.MAX_NON_SPECIAL);
THIS^.testValueIsANumber(THIS^.MIN_NON_SPECIAL);
THIS^.testValueIsANumber(THIS^.ZERO);
THIS^.testValueIsANumber(THIS^.MINUS_ZERO);
THIS^.testValueIsANumber(THIS^.MAX_SUBNORMAL);
THIS^.testValueIsANumber(THIS^.MIN_SUBNORMAL);
THIS^.testValueIsANumber(THIS^.SMALLEST_NEGATIVE_SUBNORMAL);
THIS^.testValueIsANumber(THIS^.SMALLEST_POSITIVE_SUBNORMAL);
THIS^.testValueIsANumber(THIS^.ONE_PERCENT);
THIS^.testValueIsANumber(THIS^.ONE_PERMILLE);
THIS^.testValueIsANumber(THIS^.ONE_PERCENT * -1.0);
THIS^.testValueIsANumber(THIS^.ONE_PERMILLE * -1.0);

TcUnit.TEST_FINISHED();
END_METHOD

(*

short summary
==================
This test method tests ``assert.float.single.valueIsEqualTo``
method of CNM_AssertionInterfaces library with various inputs

.. <legal notes>

legal notes
=================
| SPDX-FileCopyrightText: © 2022 ekvip automation GmbH <info@ekvip.de>
| SPDX-License-Identifier: Apache-2.0
| For details check: Apache-2.0_

.. _Apache-2.0: https://www.apache.org/licenses/LICENSE-2.0

.. </legal notes>

*)

METHOD runValueIsEqualToTests
RETURN (NOT TcUnit.TEST_ORDERED(THIS^.getTestNameFor('valueIsEqualTo')));

THIS^.testValueIsEqualTo(
	valueToTest := THIS^.NAN,
	expected := THIS^.ONE_PERCENT,
	tolerance := THIS^.ONE_PERMILLE
);

THIS^.testValueIsEqualTo(
	valueToTest := THIS^.ONE_PERCENT,
	expected := THIS^.NAN,
	tolerance := THIS^.ONE_PERMILLE
);

THIS^.testValueIsEqualTo(
	valueToTest := THIS^.ONE_PERCENT,
	expected := THIS^.ONE_PERCENT,
	tolerance := THIS^.NAN
);

THIS^.testValueIsEqualTo(
	valueToTest := THIS^.NAN,
	expected := THIS^.NAN,
	tolerance := THIS^.ONE_PERCENT
);

THIS^.testValueIsEqualTo(
	valueToTest := THIS^.NAN,
	expected := THIS^.NAN,
	tolerance := THIS^.NAN
);

THIS^.testValueIsEqualTo(
	valueToTest := THIS^.INF,
	expected := THIS^.ONE_PERCENT,
	tolerance := THIS^.ONE_PERMILLE
);

THIS^.testValueIsEqualTo(
	valueToTest := THIS^.ONE_PERCENT,
	expected := THIS^.INF,
	tolerance := THIS^.ONE_PERMILLE
);

THIS^.testValueIsEqualTo(
	valueToTest := THIS^.ONE_PERCENT,
	expected := THIS^.ONE_PERCENT,
	tolerance := THIS^.INF
);

THIS^.testValueIsEqualTo(
	valueToTest := THIS^.INF,
	expected := THIS^.INF,
	tolerance := THIS^.ONE_PERCENT
);

THIS^.testValueIsEqualTo(
	valueToTest := THIS^.INF,
	expected := THIS^.INF,
	tolerance := THIS^.INF
);

THIS^.testValueIsEqualTo(
	valueToTest := THIS^.INF,
	expected := THIS^.MINUS_INF,
	tolerance := THIS^.INF
);

THIS^.testValueIsEqualTo(
	valueToTest := THIS^.MINUS_INF,
	expected := THIS^.ONE_PERCENT,
	tolerance := THIS^.ONE_PERMILLE
);

THIS^.testValueIsEqualTo(
	valueToTest := THIS^.ONE_PERCENT,
	expected := THIS^.MINUS_INF,
	tolerance := THIS^.ONE_PERMILLE
);

THIS^.testValueIsEqualTo(
	valueToTest := THIS^.ONE_PERCENT,
	expected := THIS^.ONE_PERCENT,
	tolerance := THIS^.MINUS_INF
);

THIS^.testValueIsEqualTo(
	valueToTest := THIS^.MINUS_INF,
	expected := THIS^.MINUS_INF,
	tolerance := THIS^.ONE_PERCENT
);

THIS^.testValueIsEqualTo(
	valueToTest := THIS^.MINUS_INF,
	expected := THIS^.MINUS_INF,
	tolerance := THIS^.MINUS_INF
);

THIS^.testValueIsEqualTo(
	valueToTest := THIS^.INF,
	expected := THIS^.MINUS_INF,
	tolerance := THIS^.INF
);

THIS^.testValueIsEqualTo(
	valueToTest := THIS^.MINUS_ZERO,
	expected := THIS^.SMALLEST_POSITIVE_SUBNORMAL,
	tolerance := THIS^.ONE_PERMILLE
);

THIS^.testValueIsEqualTo(
	valueToTest := THIS^.SMALLEST_POSITIVE_SUBNORMAL,
	expected := THIS^.MINUS_ZERO,
	tolerance := THIS^.ONE_PERMILLE
);

THIS^.testValueIsEqualTo(
	valueToTest := THIS^.SMALLEST_POSITIVE_SUBNORMAL,
	expected := THIS^.SMALLEST_POSITIVE_SUBNORMAL,
	tolerance := THIS^.MINUS_ZERO
);

THIS^.testValueIsEqualTo(
	valueToTest := THIS^.MINUS_ZERO,
	expected := THIS^.MINUS_ZERO,
	tolerance := THIS^.SMALLEST_POSITIVE_SUBNORMAL
);

THIS^.testValueIsEqualTo(
	valueToTest := THIS^.MINUS_ZERO,
	expected := THIS^.MINUS_ZERO,
	tolerance := THIS^.MINUS_ZERO
);

THIS^.testValueIsEqualTo(
	valueToTest := THIS^.MINUS_ZERO,
	expected := THIS^.ZERO,
	tolerance := THIS^.MINUS_ZERO
);

THIS^.testValueIsEqualTo(
	valueToTest := THIS^.ZERO,
	expected := THIS^.SMALLEST_POSITIVE_SUBNORMAL,
	tolerance := THIS^.ONE_PERMILLE
);

THIS^.testValueIsEqualTo(
	valueToTest := THIS^.SMALLEST_POSITIVE_SUBNORMAL,
	expected := THIS^.ZERO,
	tolerance := THIS^.ONE_PERMILLE
);

THIS^.testValueIsEqualTo(
	valueToTest := THIS^.SMALLEST_POSITIVE_SUBNORMAL,
	expected := THIS^.SMALLEST_POSITIVE_SUBNORMAL,
	tolerance := THIS^.ZERO
);

THIS^.testValueIsEqualTo(
	valueToTest := THIS^.ZERO,
	expected := THIS^.ZERO,
	tolerance := THIS^.SMALLEST_POSITIVE_SUBNORMAL
);

THIS^.testValueIsEqualTo(
	valueToTest := THIS^.ZERO,
	expected := THIS^.ZERO,
	tolerance := THIS^.ZERO
);

THIS^.testValueIsEqualTo(
	valueToTest := THIS^.ZERO,
	expected := THIS^.MINUS_ZERO,
	tolerance := THIS^.ZERO
);

THIS^.testValueIsEqualTo(
	valueToTest := THIS^.SMALLEST_POSITIVE_SUBNORMAL,
	expected := THIS^.ONE_PERCENT,
	tolerance := THIS^.ONE_PERMILLE
);

THIS^.testValueIsEqualTo(
	valueToTest := THIS^.ONE_PERCENT,
	expected := THIS^.SMALLEST_POSITIVE_SUBNORMAL,
	tolerance := THIS^.ONE_PERMILLE
);

THIS^.testValueIsEqualTo(
	valueToTest := THIS^.ONE_PERCENT,
	expected := THIS^.ONE_PERCENT,
	tolerance := THIS^.SMALLEST_POSITIVE_SUBNORMAL
);

THIS^.testValueIsEqualTo(
	valueToTest := THIS^.SMALLEST_POSITIVE_SUBNORMAL,
	expected := THIS^.SMALLEST_POSITIVE_SUBNORMAL,
	tolerance := THIS^.ONE_PERCENT
);

THIS^.testValueIsEqualTo(
	valueToTest := THIS^.SMALLEST_POSITIVE_SUBNORMAL,
	expected := THIS^.SMALLEST_POSITIVE_SUBNORMAL,
	tolerance := THIS^.SMALLEST_POSITIVE_SUBNORMAL
);

THIS^.testValueIsEqualTo(
	valueToTest := THIS^.SMALLEST_POSITIVE_SUBNORMAL,
	expected := THIS^.SMALLEST_NEGATIVE_SUBNORMAL,
	tolerance := THIS^.SMALLEST_POSITIVE_SUBNORMAL
);

THIS^.testValueIsEqualTo(
	valueToTest := THIS^.SMALLEST_NEGATIVE_SUBNORMAL,
	expected := THIS^.ONE_PERCENT,
	tolerance := THIS^.ONE_PERMILLE
);

THIS^.testValueIsEqualTo(
	valueToTest := THIS^.ONE_PERCENT,
	expected := THIS^.SMALLEST_NEGATIVE_SUBNORMAL,
	tolerance := THIS^.ONE_PERMILLE
);

THIS^.testValueIsEqualTo(
	valueToTest := THIS^.ONE_PERCENT,
	expected := THIS^.ONE_PERCENT,
	tolerance := THIS^.SMALLEST_NEGATIVE_SUBNORMAL
);

THIS^.testValueIsEqualTo(
	valueToTest := THIS^.SMALLEST_NEGATIVE_SUBNORMAL,
	expected := THIS^.SMALLEST_NEGATIVE_SUBNORMAL,
	tolerance := THIS^.ONE_PERCENT
);

THIS^.testValueIsEqualTo(
	valueToTest := THIS^.SMALLEST_NEGATIVE_SUBNORMAL,
	expected := THIS^.SMALLEST_NEGATIVE_SUBNORMAL,
	tolerance := THIS^.SMALLEST_NEGATIVE_SUBNORMAL
);

THIS^.testValueIsEqualTo(
	valueToTest := THIS^.SMALLEST_NEGATIVE_SUBNORMAL,
	expected := THIS^.SMALLEST_POSITIVE_SUBNORMAL,
	tolerance := THIS^.SMALLEST_NEGATIVE_SUBNORMAL
);

THIS^.testValueIsEqualTo(
	valueToTest := THIS^.MAX_SUBNORMAL,
	expected := THIS^.SMALLEST_POSITIVE_SUBNORMAL,
	tolerance := THIS^.SMALLEST_NEGATIVE_SUBNORMAL
);

THIS^.testValueIsEqualTo(
	valueToTest := THIS^.SMALLEST_POSITIVE_SUBNORMAL,
	expected := THIS^.MAX_SUBNORMAL,
	tolerance := THIS^.SMALLEST_NEGATIVE_SUBNORMAL
);

THIS^.testValueIsEqualTo(
	valueToTest := THIS^.SMALLEST_POSITIVE_SUBNORMAL,
	expected := THIS^.SMALLEST_POSITIVE_SUBNORMAL,
	tolerance := THIS^.MAX_SUBNORMAL
);

THIS^.testValueIsEqualTo(
	valueToTest := THIS^.MAX_SUBNORMAL,
	expected := THIS^.MAX_SUBNORMAL,
	tolerance := THIS^.SMALLEST_POSITIVE_SUBNORMAL
);

THIS^.testValueIsEqualTo(
	valueToTest := THIS^.MAX_SUBNORMAL,
	expected := THIS^.MAX_SUBNORMAL,
	tolerance := THIS^.MAX_SUBNORMAL
);

THIS^.testValueIsEqualTo(
	valueToTest := THIS^.MAX_SUBNORMAL,
	expected := THIS^.MIN_SUBNORMAL,
	tolerance := THIS^.MAX_SUBNORMAL
);
//
THIS^.testValueIsEqualTo(
	valueToTest := THIS^.MIN_SUBNORMAL,
	expected := THIS^.SMALLEST_POSITIVE_SUBNORMAL,
	tolerance := THIS^.SMALLEST_NEGATIVE_SUBNORMAL
);

THIS^.testValueIsEqualTo(
	valueToTest := THIS^.SMALLEST_POSITIVE_SUBNORMAL,
	expected := THIS^.MIN_SUBNORMAL,
	tolerance := THIS^.SMALLEST_NEGATIVE_SUBNORMAL
);

THIS^.testValueIsEqualTo(
	valueToTest := THIS^.SMALLEST_POSITIVE_SUBNORMAL,
	expected := THIS^.SMALLEST_POSITIVE_SUBNORMAL,
	tolerance := THIS^.MIN_SUBNORMAL
);

THIS^.testValueIsEqualTo(
	valueToTest := THIS^.MIN_SUBNORMAL,
	expected := THIS^.MIN_SUBNORMAL,
	tolerance := THIS^.SMALLEST_POSITIVE_SUBNORMAL
);

THIS^.testValueIsEqualTo(
	valueToTest := THIS^.MIN_SUBNORMAL,
	expected := THIS^.MIN_SUBNORMAL,
	tolerance := THIS^.MIN_SUBNORMAL
);

THIS^.testValueIsEqualTo(
	valueToTest := THIS^.MIN_SUBNORMAL,
	expected := THIS^.MAX_SUBNORMAL,
	tolerance := THIS^.MIN_SUBNORMAL
);

THIS^.testValueIsEqualTo(
	valueToTest := THIS^.MAX_NON_SPECIAL,
	expected := THIS^.SMALLEST_POSITIVE_SUBNORMAL,
	tolerance := THIS^.SMALLEST_NEGATIVE_SUBNORMAL
);

THIS^.testValueIsEqualTo(
	valueToTest := THIS^.SMALLEST_POSITIVE_SUBNORMAL,
	expected := THIS^.MAX_NON_SPECIAL,
	tolerance := THIS^.SMALLEST_NEGATIVE_SUBNORMAL
);

THIS^.testValueIsEqualTo(
	valueToTest := THIS^.SMALLEST_POSITIVE_SUBNORMAL,
	expected := THIS^.SMALLEST_POSITIVE_SUBNORMAL,
	tolerance := THIS^.MAX_NON_SPECIAL
);

THIS^.testValueIsEqualTo(
	valueToTest := THIS^.MAX_NON_SPECIAL,
	expected := THIS^.MAX_NON_SPECIAL,
	tolerance := THIS^.SMALLEST_POSITIVE_SUBNORMAL
);

THIS^.testValueIsEqualTo(
	valueToTest := THIS^.MAX_NON_SPECIAL,
	expected := THIS^.MAX_NON_SPECIAL,
	tolerance := THIS^.MAX_NON_SPECIAL
);

THIS^.testValueIsEqualTo(
	valueToTest := THIS^.MAX_NON_SPECIAL,
	expected := THIS^.MIN_NON_SPECIAL,
	tolerance := THIS^.MAX_NON_SPECIAL
);

THIS^.testValueIsEqualTo(
	valueToTest := THIS^.MIN_NON_SPECIAL,
	expected := THIS^.SMALLEST_POSITIVE_SUBNORMAL,
	tolerance := THIS^.SMALLEST_NEGATIVE_SUBNORMAL
);

THIS^.testValueIsEqualTo(
	valueToTest := THIS^.SMALLEST_POSITIVE_SUBNORMAL,
	expected := THIS^.MIN_NON_SPECIAL,
	tolerance := THIS^.SMALLEST_NEGATIVE_SUBNORMAL
);

THIS^.testValueIsEqualTo(
	valueToTest := THIS^.SMALLEST_POSITIVE_SUBNORMAL,
	expected := THIS^.SMALLEST_POSITIVE_SUBNORMAL,
	tolerance := THIS^.MIN_NON_SPECIAL
);

THIS^.testValueIsEqualTo(
	valueToTest := THIS^.MIN_NON_SPECIAL,
	expected := THIS^.MIN_NON_SPECIAL,
	tolerance := THIS^.SMALLEST_POSITIVE_SUBNORMAL
);

THIS^.testValueIsEqualTo(
	valueToTest := THIS^.MIN_NON_SPECIAL,
	expected := THIS^.MIN_NON_SPECIAL,
	tolerance := THIS^.MIN_NON_SPECIAL
);

THIS^.testValueIsEqualTo(
	valueToTest := THIS^.MAX_NON_SPECIAL,
	expected := THIS^.MIN_NON_SPECIAL,
	tolerance := THIS^.MAX_NON_SPECIAL
);

TcUnit.TEST_FINISHED();
END_METHOD

(*

short summary
==================
This test method tests ``assert.float.single.valueIsFinite``
method of CNM_AssertionInterfaces library with various inputs

.. <legal notes>

legal notes
=================
| SPDX-FileCopyrightText: © 2022 ekvip automation GmbH <info@ekvip.de>
| SPDX-License-Identifier: Apache-2.0
| For details check: Apache-2.0_

.. _Apache-2.0: https://www.apache.org/licenses/LICENSE-2.0

.. </legal notes>

*)

METHOD runValueIsFiniteTests
RETURN (NOT TcUnit.TEST_ORDERED(THIS^.getTestNameFor('valueIsFinite')));

